LIN {X 0,Y 573.286,Z 595.539,A -85,B 0,C 180,E1 -2259.17,E2 -2259.17} C_VEL
LIN {X 0,Y 573.423,Z 585.099,A -85,B 0,C 180,E1 -2260.058,E2 -2260.058} C_VEL
LIN {X 0,Y 573.528,Z 573.355,A -85,B 0,C 180,E1 -2260.858,E2 -2260.858} C_VEL
LIN {X 0,Y 573.653,Z 562.283,A -85,B 0,C 180,E1 -2261.447,E2 -2261.447} C_VEL
LIN {X 0,Y 573.745,Z 549.174,A -85,B 0,C 180,E1 -2261.974,E2 -2261.974} C_VEL
LIN {X 0,Y 573.879,Z 536.521,A -85,B 0,C 180,E1 -2262.33,E2 -2262.33} C_VEL
LIN {X 0,Y 573.903,Z 523.313,A -85,B 0,C 180,E1 -2262.554,E2 -2262.554} C_VEL
LIN {X 0,Y 573.944,Z 426.723,A -85,B 0,C 180,E1 -2263.769,E2 -2263.769} C_VEL
LIN {X 0,Y 573.378,Z 422.884,A -85,B 0,C 180,E1 -2263.851,E2 -2263.851} C_VEL
LIN {X 0,Y 573.54,Z 403.262,A -85,B 0,C 180,E1 -2266.723,E2 -2266.723} C_VEL
LIN {X 0,Y 573.712,Z 385.787,A -85,B 0,C 180,E1 -2269.314,E2 -2269.314} C_VEL
LIN {X 0,Y 573.994,Z 368.402,A -85,B 0,C 180,E1 -2271.928,E2 -2271.928} C_VEL
LIN {X 0,Y 573.681,Z 364.676,A -85,B 0,C 180,E1 -2272.509,E2 -2272.509} C_VEL
LIN {X 0,Y 573.261,Z 362.581,A -85,B 0,C 180,E1 -2272.86,E2 -2272.86} C_VEL
LIN {X 0,Y 573.259,Z 362.579,A -85,B 0,C 180,E1 -2275.41,E2 -2275.41} C_VEL
LIN {X 0,Y 573.254,Z 362.574,A -85,B 0,C 180,E1 -2278.029,E2 -2278.029} C_VEL
LIN {X 0,Y 573.242,Z 362.58,A -85,B 0,C 180,E1 -2280.884,E2 -2280.884} C_VEL
LIN {X 0,Y 573.265,Z 362.574,A -85,B 0,C 180,E1 -2283.524,E2 -2283.524} C_VEL
LIN {X 0,Y 573.219,Z 362.577,A -85,B 0,C 180,E1 -2286.051,E2 -2286.051} C_VEL
LIN {X 0,Y 573.252,Z 362.577,A -85,B 0,C 180,E1 -2288.701,E2 -2288.701} C_VEL
LIN {X 0,Y 573.232,Z 362.578,A -85,B 0,C 180,E1 -2291.457,E2 -2291.457} C_VEL
LIN {X 0,Y 573.238,Z 362.576,A -85,B 0,C 180,E1 -2294.333,E2 -2294.333} C_VEL
LIN {X 0,Y 573.247,Z 362.576,A -85,B 0,C 180,E1 -2297.358,E2 -2297.358} C_VEL
LIN {X 0,Y 573.242,Z 362.577,A -85,B 0,C 180,E1 -2300.392,E2 -2300.392} C_VEL
LIN {X 0,Y 573.255,Z 362.577,A -85,B 0,C 180,E1 -2303.078,E2 -2303.078} C_VEL
LIN {X 0,Y 573.269,Z 362.57,A -85,B 0,C 180,E1 -2305.671,E2 -2305.671} C_VEL
LIN {X 0,Y 573.244,Z 362.576,A -85,B 0,C 180,E1 -2308.185,E2 -2308.185} C_VEL
LIN {X 0,Y 573.267,Z 362.58,A -85,B 0,C 180,E1 -2310.634,E2 -2310.634} C_VEL
LIN {X 0,Y 573.254,Z 362.576,A -85,B 0,C 180,E1 -2313.024,E2 -2313.024} C_VEL
LIN {X 0,Y 573.278,Z 362.57,A -85,B 0,C 180,E1 -2315.366,E2 -2315.366} C_VEL
LIN {X 0,Y 573.233,Z 362.583,A -85,B 0,C 180,E1 -2318.419,E2 -2318.419} C_VEL
LIN {X 0,Y 573.282,Z 362.575,A -85,B 0,C 180,E1 -2320.728,E2 -2320.728} C_VEL
LIN {X 0,Y 573.253,Z 362.573,A -85,B 0,C 180,E1 -2323.622,E2 -2323.622} C_VEL
LIN {X 0,Y 573.276,Z 362.571,A -85,B 0,C 180,E1 -2325.807,E2 -2325.807} C_VEL
LIN {X 0,Y 573.267,Z 362.575,A -85,B 0,C 180,E1 -2328.745,E2 -2328.745} C_VEL
LIN {X 0,Y 573.259,Z 362.572,A -85,B 0,C 180,E1 -2331.54,E2 -2331.54} C_VEL
LIN {X 0,Y 573.247,Z 362.574,A -85,B 0,C 180,E1 -2333.665,E2 -2333.665} C_VEL
LIN {X 0,Y 573.228,Z 362.578,A -85,B 0,C 180,E1 -2335.781,E2 -2335.781} C_VEL
LIN {X 0,Y 573.31,Z 362.57,A -85,B 0,C 180,E1 -2337.892,E2 -2337.892} C_VEL
LIN {X 0,Y 573.335,Z 362.565,A -85,B 0,C 180,E1 -2340.702,E2 -2340.702} C_VEL
LIN {X 0,Y 573.238,Z 362.575,A -85,B 0,C 180,E1 -2343.515,E2 -2343.515} C_VEL
LIN {X 0,Y 573.293,Z 362.57,A -85,B 0,C 180,E1 -2345.628,E2 -2345.628} C_VEL
LIN {X 0,Y 573.288,Z 362.572,A -85,B 0,C 180,E1 -2348.46,E2 -2348.46} C_VEL
LIN {X 0,Y 573.276,Z 362.57,A -85,B 0,C 180,E1 -2351.312,E2 -2351.312} C_VEL
LIN {X 0,Y 573.286,Z 362.572,A -85,B 0,C 180,E1 -2354.425,E2 -2354.425} C_VEL
LIN {X 0,Y 573.264,Z 362.571,A -85,B 0,C 180,E1 -2357.112,E2 -2357.112} C_VEL
LIN {X 0,Y 573.256,Z 362.579,A -85,B 0,C 180,E1 -2360.077,E2 -2360.077} C_VEL
LIN {X 0,Y 573.238,Z 362.575,A -85,B 0,C 180,E1 -2363.099,E2 -2363.099} C_VEL
LIN {X 0,Y 573.255,Z 362.574,A -85,B 0,C 180,E1 -2364.388,E2 -2364.388} C_VEL
LIN {X 0,Y 572.626,Z 362.652,A -85,B 0,C 180,E1 -2364.974,E2 -2364.974} C_VEL
LIN {X 0,Y 569.779,Z 363.013,A -85,B 0,C 180,E1 -2365.926,E2 -2365.926} C_VEL
LIN {X 0,Y 567.347,Z 363.315,A -85,B 0,C 180,E1 -2366.691,E2 -2366.691} C_VEL
LIN {X 0,Y 566.297,Z 363.442,A -85,B 0,C 180,E1 -2367.282,E2 -2367.282} C_VEL
LIN {X 0,Y 566.211,Z 363.452,A -85,B 0,C 180,E1 -2367.483,E2 -2367.483} C_VEL
LIN {X 0,Y 566.206,Z 363.46,A -85,B 0,C 180,E1 -2369.769,E2 -2369.769} C_VEL
LIN {X 0,Y 566.21,Z 363.45,A -85,B 0,C 180,E1 -2372.43,E2 -2372.43} C_VEL
LIN {X 0,Y 566.205,Z 363.451,A -85,B 0,C 180,E1 -2374.993,E2 -2374.993} C_VEL
LIN {X 0,Y 566.2,Z 363.458,A -85,B 0,C 180,E1 -2377.461,E2 -2377.461} C_VEL
LIN {X 0,Y 566.21,Z 363.451,A -85,B 0,C 180,E1 -2380.199,E2 -2380.199} C_VEL
LIN {X 0,Y 566.209,Z 363.453,A -85,B 0,C 180,E1 -2383.054,E2 -2383.054} C_VEL
LIN {X 0,Y 566.202,Z 363.453,A -85,B 0,C 180,E1 -2386.049,E2 -2386.049} C_VEL
LIN {X 0,Y 566.223,Z 363.454,A -85,B 0,C 180,E1 -2389.213,E2 -2389.213} C_VEL
LIN {X 0,Y 566.193,Z 363.458,A -85,B 0,C 180,E1 -2391.637,E2 -2391.637} C_VEL
LIN {X 0,Y 566.216,Z 363.449,A -85,B 0,C 180,E1 -2394.312,E2 -2394.312} C_VEL
LIN {X 0,Y 566.223,Z 363.451,A -85,B 0,C 180,E1 -2396.898,E2 -2396.898} C_VEL
LIN {X 0,Y 566.185,Z 363.461,A -85,B 0,C 180,E1 -2399.407,E2 -2399.407} C_VEL
LIN {X 0,Y 566.215,Z 363.451,A -85,B 0,C 180,E1 -2401.858,E2 -2401.858} C_VEL
LIN {X 0,Y 566.217,Z 363.45,A -85,B 0,C 180,E1 -2404.251,E2 -2404.251} C_VEL
LIN {X 0,Y 566.173,Z 363.459,A -85,B 0,C 180,E1 -2406.719,E2 -2406.719} C_VEL
LIN {X 0,Y 566.248,Z 363.457,A -85,B 0,C 180,E1 -2409.83,E2 -2409.83} C_VEL
LIN {X 0,Y 566.611,Z 367.185,A -85,B 0,C 180,E1 -2410.506,E2 -2410.506} C_VEL
LIN {X 0,Y 566.454,Z 382.099,A -85,B 0,C 180,E1 -2413.118,E2 -2413.118} C_VEL
LIN {X 0,Y 566.278,Z 399.018,A -85,B 0,C 180,E1 -2416.041,E2 -2416.041} C_VEL
LIN {X 0,Y 567.193,Z 405.355,A -85,B 0,C 180,E1 -2416.155,E2 -2416.155} C_VEL
LIN {X 0,Y 566.949,Z 505.972,A -85,B 0,C 180,E1 -2417.448,E2 -2417.448} C_VEL
LIN {X 0,Y 566.829,Z 519.227,A -85,B 0,C 180,E1 -2417.764,E2 -2417.764} C_VEL
LIN {X 0,Y 566.742,Z 531.382,A -85,B 0,C 180,E1 -2418.194,E2 -2418.194} C_VEL
LIN {X 0,Y 566.604,Z 543.662,A -85,B 0,C 180,E1 -2418.781,E2 -2418.781} C_VEL
LIN {X 0,Y 566.432,Z 555.848,A -85,B 0,C 180,E1 -2419.545,E2 -2419.545} C_VEL
LIN {X 0,Y 566.3,Z 566.133,A -85,B 0,C 180,E1 -2420.355,E2 -2420.355} C_VEL
LIN {X 0,Y 566.183,Z 575.38,A -85,B 0,C 180,E1 -2421.254,E2 -2421.254} C_VEL
LIN {X 0,Y 566.081,Z 584.35,A -85,B 0,C 180,E1 -2422.33,E2 -2422.33} C_VEL
LIN {X 0,Y 566.009,Z 591.459,A -85,B 0,C 180,E1 -2423.386,E2 -2423.386} C_VEL
LIN {X 0,Y 566.004,Z 596.452,A -85,B 0,C 180,E1 -2424.299,E2 -2424.299} C_VEL
LIN {X 0,Y 565.933,Z 601.193,A -85,B 0,C 180,E1 -2425.37,E2 -2425.37} C_VEL
LIN {X 0,Y 565.927,Z 604.826,A -85,B 0,C 180,E1 -2426.44,E2 -2426.44} C_VEL
LIN {X 0,Y 565.877,Z 606.703,A -85,B 0,C 180,E1 -2427.153,E2 -2427.153} C_VEL
LIN {X 0,Y 565.84,Z 608.128,A -85,B 0,C 180,E1 -2427.865,E2 -2427.865} C_VEL
LIN {X 0,Y 565.841,Z 609.756,A -85,B 0,C 180,E1 -2429.288,E2 -2429.288} C_VEL
LIN {X 0,Y 565.839,Z 609.996,A -85,B 0,C 180,E1 -2430,E2 -2430} C_VEL
LIN {X 0,Y 565.841,Z 609.815,A -85,B 0,C 180,E1 -2430.712,E2 -2430.712} C_VEL
LIN {X 0,Y 565.841,Z 608.268,A -85,B 0,C 180,E1 -2432.136,E2 -2432.136} C_VEL
LIN {X 0,Y 565.878,Z 606.907,A -85,B 0,C 180,E1 -2432.848,E2 -2432.848} C_VEL
LIN {X 0,Y 565.927,Z 604.029,A -85,B 0,C 180,E1 -2433.917,E2 -2433.917} C_VEL
LIN {X 0,Y 565.878,Z 600.128,A -85,B 0,C 180,E1 -2434.988,E2 -2434.988} C_VEL
LIN {X 0,Y 565.99,Z 595.096,A -85,B 0,C 180,E1 -2436.059,E2 -2436.059} C_VEL
LIN {X 0,Y 566.031,Z 588.771,A -85,B 0,C 180,E1 -2437.133,E2 -2437.133} C_VEL
LIN {X 0,Y 566.128,Z 580.848,A -85,B 0,C 180,E1 -2438.208,E2 -2438.208} C_VEL
LIN {X 0,Y 566.249,Z 570.997,A -85,B 0,C 180,E1 -2439.285,E2 -2439.285} C_VEL
LIN {X 0,Y 566.42,Z 560.677,A -85,B 0,C 180,E1 -2440.184,E2 -2440.184} C_VEL
LIN {X 0,Y 566.573,Z 549.359,A -85,B 0,C 180,E1 -2440.974,E2 -2440.974} C_VEL
LIN {X 0,Y 566.689,Z 538.183,A -85,B 0,C 180,E1 -2441.592,E2 -2441.592} C_VEL
LIN {X 0,Y 566.78,Z 525.588,A -85,B 0,C 180,E1 -2442.119,E2 -2442.119} C_VEL
LIN {X 0,Y 566.933,Z 512.409,A -85,B 0,C 180,E1 -2442.507,E2 -2442.507} C_VEL
LIN {X 0,Y 566.986,Z 500.032,A -85,B 0,C 180,E1 -2442.733,E2 -2442.733} C_VEL
LIN {X 0,Y 567.094,Z 404.105,A -85,B 0,C 180,E1 -2443.954,E2 -2443.954} C_VEL
LIN {X 0,Y 566.267,Z 399.007,A -85,B 0,C 180,E1 -2444.052,E2 -2444.052} C_VEL
LIN {X 0,Y 566.431,Z 382.626,A -85,B 0,C 180,E1 -2446.881,E2 -2446.881} C_VEL
LIN {X 0,Y 566.614,Z 367.284,A -85,B 0,C 180,E1 -2449.566,E2 -2449.566} C_VEL
LIN {X 0,Y 566.238,Z 363.454,A -85,B 0,C 180,E1 -2450.289,E2 -2450.289} C_VEL
LIN {X 0,Y 566.174,Z 363.461,A -85,B 0,C 180,E1 -2453.281,E2 -2453.281} C_VEL
LIN {X 0,Y 566.217,Z 363.451,A -85,B 0,C 180,E1 -2455.749,E2 -2455.749} C_VEL
LIN {X 0,Y 566.207,Z 363.451,A -85,B 0,C 180,E1 -2458.202,E2 -2458.202} C_VEL
LIN {X 0,Y 566.195,Z 363.457,A -85,B 0,C 180,E1 -2461.076,E2 -2461.076} C_VEL
LIN {X 0,Y 566.217,Z 363.449,A -85,B 0,C 180,E1 -2463.734,E2 -2463.734} C_VEL
LIN {X 0,Y 566.204,Z 363.458,A -85,B 0,C 180,E1 -2466.57,E2 -2466.57} C_VEL
LIN {X 0,Y 566.22,Z 363.448,A -85,B 0,C 180,E1 -2469.686,E2 -2469.686} C_VEL
LIN {X 0,Y 566.206,Z 363.455,A -85,B 0,C 180,E1 -2472.917,E2 -2472.917} C_VEL
LIN {X 0,Y 566.208,Z 363.453,A -85,B 0,C 180,E1 -2476.048,E2 -2476.048} C_VEL
LIN {X 0,Y 566.188,Z 363.457,A -85,B 0,C 180,E1 -2478.861,E2 -2478.861} C_VEL
LIN {X 0,Y 566.188,Z 363.453,A -85,B 0,C 180,E1 -2481.637,E2 -2481.637} C_VEL
LIN {X 0,Y 566.167,Z 363.463,A -85,B 0,C 180,E1 -2484.308,E2 -2484.308} C_VEL
LIN {X 0,Y 566.226,Z 363.45,A -85,B 0,C 180,E1 -2486.898,E2 -2486.898} C_VEL
LIN {X 0,Y 566.186,Z 363.453,A -85,B 0,C 180,E1 -2489.407,E2 -2489.407} C_VEL
LIN {X 0,Y 566.217,Z 363.452,A -85,B 0,C 180,E1 -2491.858,E2 -2491.858} C_VEL
LIN {X 0,Y 566.221,Z 363.459,A -85,B 0,C 180,E1 -2494.251,E2 -2494.251} C_VEL
LIN {X 0,Y 566.175,Z 363.456,A -85,B 0,C 180,E1 -2496.719,E2 -2496.719} C_VEL
LIN {X 0,Y 566.219,Z 363.451,A -85,B 0,C 180,E1 -2499.663,E2 -2499.663} C_VEL
LIN {X 0,Y 566.209,Z 363.452,A -85,B 0,C 180,E1 -2502.669,E2 -2502.669} C_VEL
LIN {X 0,Y 566.241,Z 363.449,A -85,B 0,C 180,E1 -2505.627,E2 -2505.627} C_VEL
LIN {X 0,Y 566.241,Z 363.447,A -85,B 0,C 180,E1 -2508.675,E2 -2508.675} C_VEL
LIN {X 0,Y 566.233,Z 363.449,A -85,B 0,C 180,E1 -2511.434,E2 -2511.434} C_VEL
LIN {X 0,Y 566.264,Z 363.447,A -85,B 0,C 180,E1 -2514.302,E2 -2514.302} C_VEL
LIN {X 0,Y 566.286,Z 363.451,A -85,B 0,C 180,E1 -2517.866,E2 -2517.866} C_VEL
LIN {X 0,Y 566.306,Z 363.438,A -85,B 0,C 180,E1 -2520.711,E2 -2520.711} C_VEL
LIN {X 0,Y 566.278,Z 363.441,A -85,B 0,C 180,E1 -2522.846,E2 -2522.846} C_VEL
LIN {X 0,Y 566.263,Z 363.453,A -85,B 0,C 180,E1 -2525.698,E2 -2525.698} C_VEL
LIN {X 0,Y 566.211,Z 363.45,A -85,B 0,C 180,E1 -2528.566,E2 -2528.566} C_VEL
LIN {X 0,Y 566.248,Z 363.452,A -85,B 0,C 180,E1 -2531.454,E2 -2531.454} C_VEL
LIN {X 0,Y 566.24,Z 363.446,A -85,B 0,C 180,E1 -2534.506,E2 -2534.506} C_VEL
LIN {X 0,Y 566.204,Z 363.457,A -85,B 0,C 180,E1 -2537.332,E2 -2537.332} C_VEL
LIN {X 0,Y 566.218,Z 363.449,A -85,B 0,C 180,E1 -2540.337,E2 -2540.337} C_VEL
LIN {X 0,Y 566.176,Z 363.461,A -85,B 0,C 180,E1 -2543.281,E2 -2543.281} C_VEL
LIN {X 0,Y 566.215,Z 363.454,A -85,B 0,C 180,E1 -2545.749,E2 -2545.749} C_VEL
LIN {X 0,Y 566.208,Z 363.45,A -85,B 0,C 180,E1 -2548.202,E2 -2548.202} C_VEL
LIN {X 0,Y 566.195,Z 363.457,A -85,B 0,C 180,E1 -2551.076,E2 -2551.076} C_VEL
LIN {X 0,Y 566.201,Z 363.454,A -85,B 0,C 180,E1 -2553.732,E2 -2553.732} C_VEL
LIN {X 0,Y 566.204,Z 363.452,A -85,B 0,C 180,E1 -2556.57,E2 -2556.57} C_VEL
LIN {X 0,Y 566.217,Z 363.451,A -85,B 0,C 180,E1 -2559.685,E2 -2559.685} C_VEL
LIN {X 0,Y 566.207,Z 363.456,A -85,B 0,C 180,E1 -2562.917,E2 -2562.917} C_VEL
LIN {X 0,Y 566.198,Z 363.451,A -85,B 0,C 180,E1 -2566.049,E2 -2566.049} C_VEL
LIN {X 0,Y 566.208,Z 363.457,A -85,B 0,C 180,E1 -2569.214,E2 -2569.214} C_VEL
LIN {X 0,Y 566.194,Z 363.453,A -85,B 0,C 180,E1 -2571.637,E2 -2571.637} C_VEL
LIN {X 0,Y 566.178,Z 363.455,A -85,B 0,C 180,E1 -2574.309,E2 -2574.309} C_VEL
LIN {X 0,Y 566.224,Z 363.458,A -85,B 0,C 180,E1 -2576.898,E2 -2576.898} C_VEL
LIN {X 0,Y 566.192,Z 363.455,A -85,B 0,C 180,E1 -2579.408,E2 -2579.408} C_VEL
LIN {X 0,Y 566.216,Z 363.45,A -85,B 0,C 180,E1 -2581.857,E2 -2581.857} C_VEL
LIN {X 0,Y 566.219,Z 363.453,A -85,B 0,C 180,E1 -2584.251,E2 -2584.251} C_VEL
LIN {X 0,Y 566.208,Z 363.538,A -85,B 0,C 180,E1 -2587.024,E2 -2587.024} C_VEL
LIN {X 0,Y 567.015,Z 368.31,A -85,B 0,C 180,E1 -2587.787,E2 -2587.787} C_VEL
LIN {X 0,Y 566.782,Z 385.899,A -85,B 0,C 180,E1 -2590.457,E2 -2590.457} C_VEL
LIN {X 0,Y 566.557,Z 404.552,A -85,B 0,C 180,E1 -2593.258,E2 -2593.258} C_VEL
LIN {X 0,Y 566.39,Z 423.124,A -85,B 0,C 180,E1 -2595.997,E2 -2595.997} C_VEL
LIN {X 0,Y 567.197,Z 428.387,A -85,B 0,C 180,E1 -2596.085,E2 -2596.085} C_VEL
LIN {X 0,Y 566.968,Z 530.935,A -85,B 0,C 180,E1 -2597.403,E2 -2597.403} C_VEL
LIN {X 0,Y 566.852,Z 544.211,A -85,B 0,C 180,E1 -2597.719,E2 -2597.719} C_VEL
LIN {X 0,Y 566.759,Z 556.37,A -85,B 0,C 180,E1 -2598.148,E2 -2598.148} C_VEL
LIN {X 0,Y 566.59,Z 568.445,A -85,B 0,C 180,E1 -2598.724,E2 -2598.724} C_VEL
LIN {X 0,Y 566.442,Z 580.196,A -85,B 0,C 180,E1 -2599.455,E2 -2599.455} C_VEL
LIN {X 0,Y 566.321,Z 590.599,A -85,B 0,C 180,E1 -2600.265,E2 -2600.265} C_VEL
LIN {X 0,Y 566.207,Z 599.111,A -85,B 0,C 180,E1 -2601.074,E2 -2601.074} C_VEL
LIN {X 0,Y 566.112,Z 606.959,A -85,B 0,C 180,E1 -2601.971,E2 -2601.971} C_VEL
LIN {X 0,Y 566.004,Z 614.621,A -85,B 0,C 180,E1 -2603.046,E2 -2603.046} C_VEL
LIN {X 0,Y 566.004,Z 621.679,A -85,B 0,C 180,E1 -2604.299,E2 -2604.299} C_VEL
LIN {X 0,Y 565.933,Z 626.372,A -85,B 0,C 180,E1 -2605.37,E2 -2605.37} C_VEL
LIN {X 0,Y 565.927,Z 629.957,A -85,B 0,C 180,E1 -2606.44,E2 -2606.44} C_VEL
LIN {X 0,Y 565.878,Z 631.808,A -85,B 0,C 180,E1 -2607.152,E2 -2607.152} C_VEL
LIN {X 0,Y 565.846,Z 634.185,A -85,B 0,C 180,E1 -2608.576,E2 -2608.576} C_VEL
LIN {X 0,Y 565.839,Z 635,A -85,B 0,C 180,E1 -2610,E2 -2610} C_VEL
LIN {X 0,Y 565.846,Z 634.186,A -85,B 0,C 180,E1 -2611.423,E2 -2611.423} C_VEL
LIN {X 0,Y 565.878,Z 631.81,A -85,B 0,C 180,E1 -2612.847,E2 -2612.847} C_VEL
LIN {X 0,Y 565.926,Z 628.896,A -85,B 0,C 180,E1 -2613.916,E2 -2613.916} C_VEL
LIN {X 0,Y 565.878,Z 624.949,A -85,B 0,C 180,E1 -2614.987,E2 -2614.987} C_VEL
LIN {X 0,Y 566.002,Z 619.867,A -85,B 0,C 180,E1 -2616.058,E2 -2616.058} C_VEL
LIN {X 0,Y 566.04,Z 613.469,A -85,B 0,C 180,E1 -2617.132,E2 -2617.132} C_VEL
LIN {X 0,Y 566.133,Z 605.479,A -85,B 0,C 180,E1 -2618.208,E2 -2618.208} C_VEL
LIN {X 0,Y 566.228,Z 597.336,A -85,B 0,C 180,E1 -2619.105,E2 -2619.105} C_VEL
LIN {X 0,Y 566.343,Z 587.401,A -85,B 0,C 180,E1 -2620.005,E2 -2620.005} C_VEL
LIN {X 0,Y 566.529,Z 576.292,A -85,B 0,C 180,E1 -2620.807,E2 -2620.807} C_VEL
LIN {X 0,Y 566.612,Z 565.177,A -85,B 0,C 180,E1 -2621.447,E2 -2621.447} C_VEL
LIN {X 0,Y 566.737,Z 552.984,A -85,B 0,C 180,E1 -2621.988,E2 -2621.988} C_VEL
LIN {X 0,Y 566.9,Z 540.178,A -85,B 0,C 180,E1 -2622.394,E2 -2622.394} C_VEL
LIN {X 0,Y 566.977,Z 526.605,A -85,B 0,C 180,E1 -2622.665,E2 -2622.665} C_VEL
LIN {X 0,Y 567.036,Z 427.418,A -85,B 0,C 180,E1 -2623.932,E2 -2623.932} C_VEL
LIN {X 0,Y 566.377,Z 422.884,A -85,B 0,C 180,E1 -2624.026,E2 -2624.026} C_VEL
LIN {X 0,Y 566.568,Z 402.098,A -85,B 0,C 180,E1 -2627.109,E2 -2627.109} C_VEL
LIN {X 0,Y 566.796,Z 384.545,A -85,B 0,C 180,E1 -2629.748,E2 -2629.748} C_VEL
LIN {X 0,Y 567.018,Z 368.321,A -85,B 0,C 180,E1 -2632.212,E2 -2632.212} C_VEL
LIN {X 0,Y 566.209,Z 363.46,A -85,B 0,C 180,E1 -2632.998,E2 -2632.998} C_VEL
LIN {X 0,Y 566.218,Z 363.452,A -85,B 0,C 180,E1 -2635.749,E2 -2635.749} C_VEL
LIN {X 0,Y 566.205,Z 363.452,A -85,B 0,C 180,E1 -2638.202,E2 -2638.202} C_VEL
LIN {X 0,Y 566.203,Z 363.46,A -85,B 0,C 180,E1 -2641.078,E2 -2641.078} C_VEL
LIN {X 0,Y 566.215,Z 363.45,A -85,B 0,C 180,E1 -2643.734,E2 -2643.734} C_VEL
LIN {X 0,Y 566.203,Z 363.453,A -85,B 0,C 180,E1 -2646.57,E2 -2646.57} C_VEL
LIN {X 0,Y 566.225,Z 363.453,A -85,B 0,C 180,E1 -2649.273,E2 -2649.273} C_VEL
LIN {X 0,Y 566.192,Z 363.452,A -85,B 0,C 180,E1 -2652.09,E2 -2652.09} C_VEL
LIN {X 0,Y 566.177,Z 363.462,A -85,B 0,C 180,E1 -2655.036,E2 -2655.036} C_VEL
LIN {X 0,Y 566.214,Z 363.449,A -85,B 0,C 180,E1 -2657.913,E2 -2657.913} C_VEL
LIN {X 0,Y 566.217,Z 363.457,A -85,B 0,C 180,E1 -2660.726,E2 -2660.726} C_VEL
LIN {X 0,Y 566.186,Z 363.453,A -85,B 0,C 180,E1 -2663.788,E2 -2663.788} C_VEL
LIN {X 0,Y 566.214,Z 363.452,A -85,B 0,C 180,E1 -2666.266,E2 -2666.266} C_VEL
LIN {X 0,Y 566.194,Z 363.458,A -85,B 0,C 180,E1 -2668.924,E2 -2668.924} C_VEL
LIN {X 0,Y 566.215,Z 363.45,A -85,B 0,C 180,E1 -2671.857,E2 -2671.857} C_VEL
LIN {X 0,Y 566.216,Z 363.453,A -85,B 0,C 180,E1 -2674.251,E2 -2674.251} C_VEL
LIN {X 0,Y 566.175,Z 363.462,A -85,B 0,C 180,E1 -2676.718,E2 -2676.718} C_VEL
LIN {X 0,Y 566.216,Z 363.449,A -85,B 0,C 180,E1 -2679.663,E2 -2679.663} C_VEL
LIN {X 0,Y 566.202,Z 363.458,A -85,B 0,C 180,E1 -2682.668,E2 -2682.668} C_VEL
LIN {X 0,Y 566.237,Z 363.447,A -85,B 0,C 180,E1 -2685.627,E2 -2685.627} C_VEL
LIN {X 0,Y 566.239,Z 363.451,A -85,B 0,C 180,E1 -2688.675,E2 -2688.675} C_VEL
LIN {X 0,Y 566.209,Z 363.45,A -85,B 0,C 180,E1 -2691.434,E2 -2691.434} C_VEL
LIN {X 0,Y 566.259,Z 363.454,A -85,B 0,C 180,E1 -2694.302,E2 -2694.302} C_VEL
LIN {X 0,Y 566.282,Z 363.445,A -85,B 0,C 180,E1 -2697.866,E2 -2697.866} C_VEL
LIN {X 0,Y 566.305,Z 363.44,A -85,B 0,C 180,E1 -2700.711,E2 -2700.711} C_VEL
LIN {X 0,Y 566.277,Z 363.442,A -85,B 0,C 180,E1 -2702.846,E2 -2702.846} C_VEL
LIN {X 0,Y 566.261,Z 363.447,A -85,B 0,C 180,E1 -2705.698,E2 -2705.698} C_VEL
LIN {X 0,Y 566.231,Z 363.45,A -85,B 0,C 180,E1 -2708.566,E2 -2708.566} C_VEL
LIN {X 0,Y 566.246,Z 363.447,A -85,B 0,C 180,E1 -2711.454,E2 -2711.454} C_VEL
LIN {X 0,Y 566.239,Z 363.448,A -85,B 0,C 180,E1 -2714.507,E2 -2714.507} C_VEL
LIN {X 0,Y 566.208,Z 363.452,A -85,B 0,C 180,E1 -2717.331,E2 -2717.331} C_VEL
LIN {X 0,Y 566.217,Z 363.452,A -85,B 0,C 180,E1 -2720.337,E2 -2720.337} C_VEL
LIN {X 0,Y 566.193,Z 363.455,A -85,B 0,C 180,E1 -2723.404,E2 -2723.404} C_VEL
LIN {X 0,Y 566.22,Z 363.458,A -85,B 0,C 180,E1 -2725.749,E2 -2725.749} C_VEL
LIN {X 0,Y 566.211,Z 363.452,A -85,B 0,C 180,E1 -2727.483,E2 -2727.483} C_VEL
LIN {X 0,Y 565.538,Z 363.539,A -85,B 0,C 180,E1 -2728.076,E2 -2728.076} C_VEL
LIN {X 0,Y 562.671,Z 363.892,A -85,B 0,C 180,E1 -2729.04,E2 -2729.04} C_VEL
LIN {X 0,Y 560.256,Z 364.2,A -85,B 0,C 180,E1 -2729.815,E2 -2729.815} C_VEL
LIN {X 0,Y 559.226,Z 364.322,A -85,B 0,C 180,E1 -2730.414,E2 -2730.414} C_VEL
LIN {X 0,Y 559.146,Z 364.33,A -85,B 0,C 180,E1 -2730.617,E2 -2730.617} C_VEL
LIN {X 0,Y 559.168,Z 364.335,A -85,B 0,C 180,E1 -2733.575,E2 -2733.575} C_VEL
LIN {X 0,Y 559.171,Z 364.327,A -85,B 0,C 180,E1 -2736.448,E2 -2736.448} C_VEL
LIN {X 0,Y 559.178,Z 364.327,A -85,B 0,C 180,E1 -2738.934,E2 -2738.934} C_VEL
LIN {X 0,Y 559.181,Z 364.327,A -85,B 0,C 180,E1 -2742.138,E2 -2742.138} C_VEL
LIN {X 0,Y 559.144,Z 364.33,A -85,B 0,C 180,E1 -2744.739,E2 -2744.739} C_VEL
LIN {X 0,Y 559.161,Z 364.334,A -85,B 0,C 180,E1 -2747.256,E2 -2747.256} C_VEL
LIN {X 0,Y 559.185,Z 364.326,A -85,B 0,C 180,E1 -2750.135,E2 -2750.135} C_VEL
LIN {X 0,Y 559.15,Z 364.332,A -85,B 0,C 180,E1 -2752.892,E2 -2752.892} C_VEL
LIN {X 0,Y 559.161,Z 364.334,A -85,B 0,C 180,E1 -2755.556,E2 -2755.556} C_VEL
LIN {X 0,Y 559.169,Z 364.327,A -85,B 0,C 180,E1 -2758.137,E2 -2758.137} C_VEL
LIN {X 0,Y 559.146,Z 364.331,A -85,B 0,C 180,E1 -2760.646,E2 -2760.646} C_VEL
LIN {X 0,Y 559.174,Z 364.335,A -85,B 0,C 180,E1 -2763.173,E2 -2763.173} C_VEL
LIN {X 0,Y 559.159,Z 364.335,A -85,B 0,C 180,E1 -2765.495,E2 -2765.495} C_VEL
LIN {X 0,Y 559.175,Z 364.331,A -85,B 0,C 180,E1 -2768.624,E2 -2768.624} C_VEL
LIN {X 0,Y 559.211,Z 364.505,A -85,B 0,C 180,E1 -2769.733,E2 -2769.733} C_VEL
LIN {X 0,Y 559.644,Z 367.893,A -85,B 0,C 180,E1 -2770.365,E2 -2770.365} C_VEL
LIN {X 0,Y 559.447,Z 382.395,A -85,B 0,C 180,E1 -2772.952,E2 -2772.952} C_VEL
LIN {X 0,Y 559.25,Z 399.021,A -85,B 0,C 180,E1 -2775.861,E2 -2775.861} C_VEL
LIN {X 0,Y 560.276,Z 405.401,A -85,B 0,C 180,E1 -2775.981,E2 -2775.981} C_VEL
LIN {X 0,Y 560.047,Z 506,A -85,B 0,C 180,E1 -2777.291,E2 -2777.291} C_VEL
LIN {X 0,Y 559.91,Z 519.245,A -85,B 0,C 180,E1 -2777.61,E2 -2777.61} C_VEL
LIN {X 0,Y 559.786,Z 531.397,A -85,B 0,C 180,E1 -2778.045,E2 -2778.045} C_VEL
LIN {X 0,Y 559.649,Z 543.084,A -85,B 0,C 180,E1 -2778.607,E2 -2778.607} C_VEL
LIN {X 0,Y 559.481,Z 554.564,A -85,B 0,C 180,E1 -2779.322,E2 -2779.322} C_VEL
LIN {X 0,Y 559.307,Z 565.081,A -85,B 0,C 180,E1 -2780.142,E2 -2780.142} C_VEL
LIN {X 0,Y 559.197,Z 573.676,A -85,B 0,C 180,E1 -2780.961,E2 -2780.961} C_VEL
LIN {X 0,Y 559.05,Z 581.596,A -85,B 0,C 180,E1 -2781.87,E2 -2781.87} C_VEL
LIN {X 0,Y 558.971,Z 589.457,A -85,B 0,C 180,E1 -2782.977,E2 -2782.977} C_VEL
LIN {X 0,Y 558.936,Z 596.455,A -85,B 0,C 180,E1 -2784.227,E2 -2784.227} C_VEL
LIN {X 0,Y 558.827,Z 601.195,A -85,B 0,C 180,E1 -2785.311,E2 -2785.311} C_VEL
LIN {X 0,Y 558.836,Z 604.828,A -85,B 0,C 180,E1 -2786.395,E2 -2786.395} C_VEL
LIN {X 0,Y 558.799,Z 606.704,A -85,B 0,C 180,E1 -2787.116,E2 -2787.116} C_VEL
LIN {X 0,Y 558.746,Z 608.128,A -85,B 0,C 180,E1 -2787.838,E2 -2787.838} C_VEL
LIN {X 0,Y 558.741,Z 609.757,A -85,B 0,C 180,E1 -2789.279,E2 -2789.279} C_VEL
LIN {X 0,Y 558.74,Z 609.996,A -85,B 0,C 180,E1 -2790,E2 -2790} C_VEL
LIN {X 0,Y 558.741,Z 609.815,A -85,B 0,C 180,E1 -2790.721,E2 -2790.721} C_VEL
LIN {X 0,Y 558.746,Z 608.266,A -85,B 0,C 180,E1 -2792.163,E2 -2792.163} C_VEL
LIN {X 0,Y 558.8,Z 606.905,A -85,B 0,C 180,E1 -2792.884,E2 -2792.884} C_VEL
LIN {X 0,Y 558.844,Z 604.027,A -85,B 0,C 180,E1 -2793.966,E2 -2793.966} C_VEL
LIN {X 0,Y 558.798,Z 600.126,A -85,B 0,C 180,E1 -2795.051,E2 -2795.051} C_VEL
LIN {X 0,Y 558.91,Z 595.093,A -85,B 0,C 180,E1 -2796.136,E2 -2796.136} C_VEL
LIN {X 0,Y 558.973,Z 588.767,A -85,B 0,C 180,E1 -2797.223,E2 -2797.223} C_VEL
LIN {X 0,Y 559.091,Z 580.843,A -85,B 0,C 180,E1 -2798.312,E2 -2798.312} C_VEL
LIN {X 0,Y 559.224,Z 570.99,A -85,B 0,C 180,E1 -2799.403,E2 -2799.403} C_VEL
LIN {X 0,Y 559.412,Z 560.67,A -85,B 0,C 180,E1 -2800.313,E2 -2800.313} C_VEL
LIN {X 0,Y 559.588,Z 549.687,A -85,B 0,C 180,E1 -2801.091,E2 -2801.091} C_VEL
LIN {X 0,Y 559.725,Z 538.171,A -85,B 0,C 180,E1 -2801.738,E2 -2801.738} C_VEL
LIN {X 0,Y 559.83,Z 525.571,A -85,B 0,C 180,E1 -2802.272,E2 -2802.272} C_VEL
LIN {X 0,Y 560.015,Z 512.385,A -85,B 0,C 180,E1 -2802.664,E2 -2802.664} C_VEL
LIN {X 0,Y 560.088,Z 499.989,A -85,B 0,C 180,E1 -2802.893,E2 -2802.893} C_VEL
LIN {X 0,Y 560.254,Z 405.177,A -85,B 0,C 180,E1 -2804.113,E2 -2804.113} C_VEL
LIN {X 0,Y 559.248,Z 399.003,A -85,B 0,C 180,E1 -2804.232,E2 -2804.232} C_VEL
LIN {X 0,Y 559.438,Z 381.481,A -85,B 0,C 180,E1 -2807.3,E2 -2807.3} C_VEL
LIN {X 0,Y 559.627,Z 367.376,A -85,B 0,C 180,E1 -2809.821,E2 -2809.821} C_VEL
LIN {X 0,Y 559.188,Z 364.333,A -85,B 0,C 180,E1 -2810.412,E2 -2810.412} C_VEL
LIN {X 0,Y 559.143,Z 364.335,A -85,B 0,C 180,E1 -2813.428,E2 -2813.428} C_VEL
LIN {X 0,Y 559.184,Z 364.328,A -85,B 0,C 180,E1 -2816.097,E2 -2816.097} C_VEL
LIN {X 0,Y 559.168,Z 364.332,A -85,B 0,C 180,E1 -2818.53,E2 -2818.53} C_VEL
LIN {X 0,Y 559.15,Z 364.332,A -85,B 0,C 180,E1 -2821.273,E2 -2821.273} C_VEL
LIN {X 0,Y 559.172,Z 364.327,A -85,B 0,C 180,E1 -2823.95,E2 -2823.95} C_VEL
LIN {X 0,Y 559.145,Z 364.333,A -85,B 0,C 180,E1 -2827.109,E2 -2827.109} C_VEL
LIN {X 0,Y 559.166,Z 364.328,A -85,B 0,C 180,E1 -2829.942,E2 -2829.942} C_VEL
LIN {X 0,Y 559.162,Z 364.335,A -85,B 0,C 180,E1 -2832.744,E2 -2832.744} C_VEL
LIN {X 0,Y 559.161,Z 364.328,A -85,B 0,C 180,E1 -2835.761,E2 -2835.761} C_VEL
LIN {X 0,Y 559.194,Z 364.329,A -85,B 0,C 180,E1 -2838.232,E2 -2838.232} C_VEL
LIN {X 0,Y 559.178,Z 364.326,A -85,B 0,C 180,E1 -2841.192,E2 -2841.192} C_VEL
LIN {X 0,Y 559.144,Z 364.331,A -85,B 0,C 180,E1 -2843.789,E2 -2843.789} C_VEL
LIN {X 0,Y 559.168,Z 364.336,A -85,B 0,C 180,E1 -2846.425,E2 -2846.425} C_VEL
LIN {X 0,Y 559.161,Z 364.329,A -85,B 0,C 180,E1 -2848.981,E2 -2848.981} C_VEL
LIN {X 0,Y 559.174,Z 364.327,A -85,B 0,C 180,E1 -2851.619,E2 -2851.619} C_VEL
LIN {X 0,Y 559.188,Z 364.329,A -85,B 0,C 180,E1 -2853.903,E2 -2853.903} C_VEL
LIN {X 0,Y 559.145,Z 364.334,A -85,B 0,C 180,E1 -2856.572,E2 -2856.572} C_VEL
LIN {X 0,Y 559.186,Z 364.325,A -85,B 0,C 180,E1 -2859.396,E2 -2859.396} C_VEL
LIN {X 0,Y 559.155,Z 364.332,A -85,B 0,C 180,E1 -2861.686,E2 -2861.686} C_VEL
LIN {X 0,Y 559.17,Z 364.334,A -85,B 0,C 180,E1 -2863.948,E2 -2863.948} C_VEL
LIN {X 0,Y 559.178,Z 364.333,A -85,B 0,C 180,E1 -2866.184,E2 -2866.184} C_VEL
LIN {X 0,Y 559.201,Z 364.323,A -85,B 0,C 180,E1 -2869.134,E2 -2869.134} C_VEL
LIN {X 0,Y 559.21,Z 364.33,A -85,B 0,C 180,E1 -2872.054,E2 -2872.054} C_VEL
LIN {X 0,Y 559.258,Z 364.316,A -85,B 0,C 180,E1 -2874.953,E2 -2874.953} C_VEL
LIN {X 0,Y 559.257,Z 364.326,A -85,B 0,C 180,E1 -2877.839,E2 -2877.839} C_VEL
LIN {X 0,Y 559.277,Z 364.314,A -85,B 0,C 180,E1 -2880.72,E2 -2880.72} C_VEL
LIN {X 0,Y 559.244,Z 364.318,A -85,B 0,C 180,E1 -2882.881,E2 -2882.881} C_VEL
LIN {X 0,Y 559.233,Z 364.328,A -85,B 0,C 180,E1 -2885.77,E2 -2885.77} C_VEL
LIN {X 0,Y 559.175,Z 364.326,A -85,B 0,C 180,E1 -2888.675,E2 -2888.675} C_VEL
LIN {X 0,Y 559.211,Z 364.331,A -85,B 0,C 180,E1 -2891.6,E2 -2891.6} C_VEL
LIN {X 0,Y 559.206,Z 364.322,A -85,B 0,C 180,E1 -2894.595,E2 -2894.595} C_VEL
LIN {X 0,Y 559.163,Z 364.338,A -85,B 0,C 180,E1 -2897.557,E2 -2897.557} C_VEL
LIN {X 0,Y 559.175,Z 364.331,A -85,B 0,C 180,E1 -2899.837,E2 -2899.837} C_VEL
LIN {X 0,Y 559.147,Z 364.331,A -85,B 0,C 180,E1 -2902.153,E2 -2902.153} C_VEL
LIN {X 0,Y 559.181,Z 364.333,A -85,B 0,C 180,E1 -2905.298,E2 -2905.298} C_VEL
LIN {X 0,Y 559.173,Z 364.326,A -85,B 0,C 180,E1 -2908.381,E2 -2908.381} C_VEL
LIN {X 0,Y 559.151,Z 364.338,A -85,B 0,C 180,E1 -2911.273,E2 -2911.273} C_VEL
LIN {X 0,Y 559.159,Z 364.329,A -85,B 0,C 180,E1 -2913.947,E2 -2913.947} C_VEL
LIN {X 0,Y 559.145,Z 364.338,A -85,B 0,C 180,E1 -2917.108,E2 -2917.108} C_VEL
LIN {X 0,Y 559.164,Z 364.328,A -85,B 0,C 180,E1 -2919.941,E2 -2919.941} C_VEL
LIN {X 0,Y 559.163,Z 364.331,A -85,B 0,C 180,E1 -2922.743,E2 -2922.743} C_VEL
LIN {X 0,Y 559.153,Z 364.33,A -85,B 0,C 180,E1 -2925.761,E2 -2925.761} C_VEL
LIN {X 0,Y 559.166,Z 364.327,A -85,B 0,C 180,E1 -2928.23,E2 -2928.23} C_VEL
LIN {X 0,Y 559.182,Z 364.332,A -85,B 0,C 180,E1 -2931.191,E2 -2931.191} C_VEL
LIN {X 0,Y 559.145,Z 364.33,A -85,B 0,C 180,E1 -2933.789,E2 -2933.789} C_VEL
LIN {X 0,Y 559.167,Z 364.33,A -85,B 0,C 180,E1 -2936.425,E2 -2936.425} C_VEL
LIN {X 0,Y 559.167,Z 364.336,A -85,B 0,C 180,E1 -2938.981,E2 -2938.981} C_VEL
LIN {X 0,Y 559.172,Z 364.328,A -85,B 0,C 180,E1 -2941.619,E2 -2941.619} C_VEL
LIN {X 0,Y 559.186,Z 364.327,A -85,B 0,C 180,E1 -2943.903,E2 -2943.903} C_VEL
LIN {X 0,Y 559.199,Z 364.482,A -85,B 0,C 180,E1 -2946.888,E2 -2946.888} C_VEL
LIN {X 0,Y 560.066,Z 369.428,A -85,B 0,C 180,E1 -2947.691,E2 -2947.691} C_VEL
LIN {X 0,Y 559.811,Z 387.353,A -85,B 0,C 180,E1 -2950.434,E2 -2950.434} C_VEL
LIN {X 0,Y 559.586,Z 403.777,A -85,B 0,C 180,E1 -2952.926,E2 -2952.926} C_VEL
LIN {X 0,Y 559.369,Z 423.124,A -85,B 0,C 180,E1 -2955.818,E2 -2955.818} C_VEL
LIN {X 0,Y 560.303,Z 430.279,A -85,B 0,C 180,E1 -2955.935,E2 -2955.935} C_VEL
LIN {X 0,Y 560.049,Z 530.935,A -85,B 0,C 180,E1 -2957.245,E2 -2957.245} C_VEL
LIN {X 0,Y 559.939,Z 544.21,A -85,B 0,C 180,E1 -2957.565,E2 -2957.565} C_VEL
LIN {X 0,Y 559.809,Z 556.372,A -85,B 0,C 180,E1 -2957.999,E2 -2957.999} C_VEL
LIN {X 0,Y 559.616,Z 568.315,A -85,B 0,C 180,E1 -2958.574,E2 -2958.574} C_VEL
LIN {X 0,Y 559.462,Z 580.194,A -85,B 0,C 180,E1 -2959.322,E2 -2959.322} C_VEL
LIN {X 0,Y 559.302,Z 590.601,A -85,B 0,C 180,E1 -2960.142,E2 -2960.142} C_VEL
LIN {X 0,Y 559.162,Z 599.111,A -85,B 0,C 180,E1 -2960.961,E2 -2960.961} C_VEL
LIN {X 0,Y 559.05,Z 606.959,A -85,B 0,C 180,E1 -2961.869,E2 -2961.869} C_VEL
LIN {X 0,Y 558.944,Z 614.621,A -85,B 0,C 180,E1 -2962.958,E2 -2962.958} C_VEL
LIN {X 0,Y 558.935,Z 621.679,A -85,B 0,C 180,E1 -2964.227,E2 -2964.227} C_VEL
LIN {X 0,Y 558.827,Z 626.372,A -85,B 0,C 180,E1 -2965.311,E2 -2965.311} C_VEL
LIN {X 0,Y 558.836,Z 629.957,A -85,B 0,C 180,E1 -2966.395,E2 -2966.395} C_VEL
LIN {X 0,Y 558.799,Z 631.807,A -85,B 0,C 180,E1 -2967.116,E2 -2967.116} C_VEL
LIN {X 0,Y 558.745,Z 634.184,A -85,B 0,C 180,E1 -2968.558,E2 -2968.558} C_VEL
LIN {X 0,Y 558.74,Z 635,A -85,B 0,C 180,E1 -2970,E2 -2970} C_VEL
LIN {X 0,Y 558.745,Z 634.185,A -85,B 0,C 180,E1 -2971.441,E2 -2971.441} C_VEL
LIN {X 0,Y 558.799,Z 631.81,A -85,B 0,C 180,E1 -2972.884,E2 -2972.884} C_VEL
LIN {X 0,Y 558.843,Z 628.896,A -85,B 0,C 180,E1 -2973.966,E2 -2973.966} C_VEL
LIN {X 0,Y 558.799,Z 624.949,A -85,B 0,C 180,E1 -2975.051,E2 -2975.051} C_VEL
LIN {X 0,Y 558.921,Z 619.867,A -85,B 0,C 180,E1 -2976.135,E2 -2976.135} C_VEL
LIN {X 0,Y 558.977,Z 613.468,A -85,B 0,C 180,E1 -2977.223,E2 -2977.223} C_VEL
LIN {X 0,Y 559.099,Z 605.478,A -85,B 0,C 180,E1 -2978.312,E2 -2978.312} C_VEL
LIN {X 0,Y 559.184,Z 597.335,A -85,B 0,C 180,E1 -2979.221,E2 -2979.221} C_VEL
LIN {X 0,Y 559.356,Z 587.4,A -85,B 0,C 180,E1 -2980.131,E2 -2980.131} C_VEL
LIN {X 0,Y 559.543,Z 576.4,A -85,B 0,C 180,E1 -2980.937,E2 -2980.937} C_VEL
LIN {X 0,Y 559.671,Z 564.461,A -85,B 0,C 180,E1 -2981.628,E2 -2981.628} C_VEL
LIN {X 0,Y 559.82,Z 551.769,A -85,B 0,C 180,E1 -2982.185,E2 -2982.185} C_VEL
LIN {X 0,Y 560.009,Z 538.348,A -85,B 0,C 180,E1 -2982.595,E2 -2982.595} C_VEL
LIN {X 0,Y 560.087,Z 525.088,A -85,B 0,C 180,E1 -2982.846,E2 -2982.846} C_VEL
LIN {X 0,Y 560.189,Z 428.412,A -85,B 0,C 180,E1 -2984.092,E2 -2984.092} C_VEL
LIN {X 0,Y 559.37,Z 422.884,A -85,B 0,C 180,E1 -2984.205,E2 -2984.205} C_VEL
LIN {X 0,Y 559.625,Z 401.877,A -85,B 0,C 180,E1 -2987.361,E2 -2987.361} C_VEL
LIN {X 0,Y 559.947,Z 380.727,A -85,B 0,C 180,E1 -2990.575,E2 -2990.575} C_VEL
LIN {X 0,Y 560.067,Z 369.45,A -85,B 0,C 180,E1 -2992.308,E2 -2992.308} C_VEL
LIN {X 0,Y 559.169,Z 364.337,A -85,B 0,C 180,E1 -2993.149,E2 -2993.149} C_VEL
LIN {X 0,Y 559.185,Z 364.326,A -85,B 0,C 180,E1 -2996.097,E2 -2996.097} C_VEL
LIN {X 0,Y 559.166,Z 364.33,A -85,B 0,C 180,E1 -2998.53,E2 -2998.53} C_VEL
LIN {X 0,Y 559.157,Z 364.336,A -85,B 0,C 180,E1 -3001.275,E2 -3001.275} C_VEL
LIN {X 0,Y 559.17,Z 364.327,A -85,B 0,C 180,E1 -3003.949,E2 -3003.949} C_VEL
LIN {X 0,Y 559.144,Z 364.339,A -85,B 0,C 180,E1 -3007.108,E2 -3007.108} C_VEL
LIN {X 0,Y 559.168,Z 364.327,A -85,B 0,C 180,E1 -3009.942,E2 -3009.942} C_VEL
LIN {X 0,Y 559.16,Z 364.334,A -85,B 0,C 180,E1 -3012.744,E2 -3012.744} C_VEL
LIN {X 0,Y 559.159,Z 364.328,A -85,B 0,C 180,E1 -3015.76,E2 -3015.76} C_VEL
LIN {X 0,Y 559.19,Z 364.326,A -85,B 0,C 180,E1 -3018.232,E2 -3018.232} C_VEL
LIN {X 0,Y 559.177,Z 364.33,A -85,B 0,C 180,E1 -3021.192,E2 -3021.192} C_VEL
LIN {X 0,Y 559.141,Z 364.33,A -85,B 0,C 180,E1 -3023.789,E2 -3023.789} C_VEL
LIN {X 0,Y 559.166,Z 364.332,A -85,B 0,C 180,E1 -3026.425,E2 -3026.425} C_VEL
LIN {X 0,Y 559.158,Z 364.333,A -85,B 0,C 180,E1 -3028.981,E2 -3028.981} C_VEL
LIN {X 0,Y 559.171,Z 364.327,A -85,B 0,C 180,E1 -3031.619,E2 -3031.619} C_VEL
LIN {X 0,Y 559.183,Z 364.326,A -85,B 0,C 180,E1 -3033.903,E2 -3033.903} C_VEL
LIN {X 0,Y 559.145,Z 364.34,A -85,B 0,C 180,E1 -3036.571,E2 -3036.571} C_VEL
LIN {X 0,Y 559.183,Z 364.325,A -85,B 0,C 180,E1 -3039.396,E2 -3039.396} C_VEL
LIN {X 0,Y 559.144,Z 364.33,A -85,B 0,C 180,E1 -3041.686,E2 -3041.686} C_VEL
LIN {X 0,Y 559.169,Z 364.329,A -85,B 0,C 180,E1 -3043.948,E2 -3043.948} C_VEL
LIN {X 0,Y 559.174,Z 364.332,A -85,B 0,C 180,E1 -3046.184,E2 -3046.184} C_VEL
LIN {X 0,Y 559.197,Z 364.324,A -85,B 0,C 180,E1 -3049.134,E2 -3049.134} C_VEL
LIN {X 0,Y 559.199,Z 364.328,A -85,B 0,C 180,E1 -3052.054,E2 -3052.054} C_VEL
LIN {X 0,Y 559.256,Z 364.317,A -85,B 0,C 180,E1 -3054.953,E2 -3054.953} C_VEL
LIN {X 0,Y 559.253,Z 364.32,A -85,B 0,C 180,E1 -3057.839,E2 -3057.839} C_VEL
LIN {X 0,Y 559.276,Z 364.316,A -85,B 0,C 180,E1 -3060.72,E2 -3060.72} C_VEL
LIN {X 0,Y 559.243,Z 364.318,A -85,B 0,C 180,E1 -3062.881,E2 -3062.881} C_VEL
LIN {X 0,Y 559.231,Z 364.323,A -85,B 0,C 180,E1 -3065.77,E2 -3065.77} C_VEL
LIN {X 0,Y 559.19,Z 364.326,A -85,B 0,C 180,E1 -3068.674,E2 -3068.674} C_VEL
LIN {X 0,Y 559.21,Z 364.325,A -85,B 0,C 180,E1 -3071.6,E2 -3071.6} C_VEL
LIN {X 0,Y 559.204,Z 364.324,A -85,B 0,C 180,E1 -3074.596,E2 -3074.596} C_VEL
LIN {X 0,Y 559.167,Z 364.331,A -85,B 0,C 180,E1 -3077.557,E2 -3077.557} C_VEL
LIN {X 0,Y 559.176,Z 364.335,A -85,B 0,C 180,E1 -3079.837,E2 -3079.837} C_VEL
LIN {X 0,Y 559.146,Z 364.335,A -85,B 0,C 180,E1 -3082.153,E2 -3082.153} C_VEL
LIN {X 0,Y 559.183,Z 364.326,A -85,B 0,C 180,E1 -3085.187,E2 -3085.187} C_VEL
LIN {X 0,Y 559.193,Z 364.333,A -85,B 0,C 180,E1 -3087.712,E2 -3087.712} C_VEL
LIN {X 0,Y 559.146,Z 364.33,A -85,B 0,C 180,E1 -3090.617,E2 -3090.617} C_VEL
LIN {X 0,Y 558.486,Z 364.416,A -85,B 0,C 180,E1 -3091.218,E2 -3091.218} C_VEL
LIN {X 0,Y 555.626,Z 364.771,A -85,B 0,C 180,E1 -3092.195,E2 -3092.195} C_VEL
LIN {X 0,Y 553.213,Z 365.07,A -85,B 0,C 180,E1 -3092.98,E2 -3092.98} C_VEL
LIN {X 0,Y 552.192,Z 365.204,A -85,B 0,C 180,E1 -3093.587,E2 -3093.587} C_VEL
LIN {X 0,Y 552.117,Z 365.207,A -85,B 0,C 180,E1 -3093.792,E2 -3093.792} C_VEL
LIN {X 0,Y 552.115,Z 365.206,A -85,B 0,C 180,E1 -3096.747,E2 -3096.747} C_VEL
LIN {X 0,Y 552.133,Z 365.212,A -85,B 0,C 180,E1 -3099.527,E2 -3099.527} C_VEL
LIN {X 0,Y 552.134,Z 365.203,A -85,B 0,C 180,E1 -3102.425,E2 -3102.425} C_VEL
LIN {X 0,Y 552.102,Z 365.216,A -85,B 0,C 180,E1 -3105.563,E2 -3105.563} C_VEL
LIN {X 0,Y 552.135,Z 365.204,A -85,B 0,C 180,E1 -3108.677,E2 -3108.677} C_VEL
LIN {X 0,Y 552.123,Z 365.215,A -85,B 0,C 180,E1 -3111.411,E2 -3111.411} C_VEL
LIN {X 0,Y 552.117,Z 365.206,A -85,B 0,C 180,E1 -3114.159,E2 -3114.159} C_VEL
LIN {X 0,Y 552.119,Z 365.207,A -85,B 0,C 180,E1 -3116.814,E2 -3116.814} C_VEL
LIN {X 0,Y 552.106,Z 365.215,A -85,B 0,C 180,E1 -3119.391,E2 -3119.391} C_VEL
LIN {X 0,Y 552.112,Z 365.207,A -85,B 0,C 180,E1 -3121.902,E2 -3121.902} C_VEL
LIN {X 0,Y 552.159,Z 365.203,A -85,B 0,C 180,E1 -3124.65,E2 -3124.65} C_VEL
LIN {X 0,Y 552.095,Z 365.215,A -85,B 0,C 180,E1 -3127.549,E2 -3127.549} C_VEL
LIN {X 0,Y 552.16,Z 365.289,A -85,B 0,C 180,E1 -3129.584,E2 -3129.584} C_VEL
LIN {X 0,Y 552.65,Z 369.95,A -85,B 0,C 180,E1 -3130.46,E2 -3130.46} C_VEL
LIN {X 0,Y 552.451,Z 384.971,A -85,B 0,C 180,E1 -3133.177,E2 -3133.177} C_VEL
LIN {X 0,Y 552.237,Z 399.236,A -85,B 0,C 180,E1 -3135.69,E2 -3135.69} C_VEL
LIN {X 0,Y 553.414,Z 406.711,A -85,B 0,C 180,E1 -3135.82,E2 -3135.82} C_VEL
LIN {X 0,Y 553.144,Z 506.029,A -85,B 0,C 180,E1 -3137.13,E2 -3137.13} C_VEL
LIN {X 0,Y 552.994,Z 519.263,A -85,B 0,C 180,E1 -3137.453,E2 -3137.453} C_VEL
LIN {X 0,Y 552.837,Z 531.411,A -85,B 0,C 180,E1 -3137.892,E2 -3137.892} C_VEL
LIN {X 0,Y 552.688,Z 542.906,A -85,B 0,C 180,E1 -3138.451,E2 -3138.451} C_VEL
LIN {X 0,Y 552.506,Z 554.57,A -85,B 0,C 180,E1 -3139.186,E2 -3139.186} C_VEL
LIN {X 0,Y 552.305,Z 565.086,A -85,B 0,C 180,E1 -3140.016,E2 -3140.016} C_VEL
LIN {X 0,Y 552.153,Z 573.681,A -85,B 0,C 180,E1 -3140.845,E2 -3140.845} C_VEL
LIN {X 0,Y 552.007,Z 581.6,A -85,B 0,C 180,E1 -3141.765,E2 -3141.765} C_VEL
LIN {X 0,Y 551.895,Z 589.461,A -85,B 0,C 180,E1 -3142.886,E2 -3142.886} C_VEL
LIN {X 0,Y 551.868,Z 596.457,A -85,B 0,C 180,E1 -3144.153,E2 -3144.153} C_VEL
LIN {X 0,Y 551.725,Z 601.198,A -85,B 0,C 180,E1 -3145.251,E2 -3145.251} C_VEL
LIN {X 0,Y 551.75,Z 604.83,A -85,B 0,C 180,E1 -3146.349,E2 -3146.349} C_VEL
LIN {X 0,Y 551.723,Z 606.706,A -85,B 0,C 180,E1 -3147.079,E2 -3147.079} C_VEL
LIN {X 0,Y 551.657,Z 608.128,A -85,B 0,C 180,E1 -3147.81,E2 -3147.81} C_VEL
LIN {X 0,Y 551.642,Z 609.757,A -85,B 0,C 180,E1 -3149.27,E2 -3149.27} C_VEL
LIN {X 0,Y 551.641,Z 609.996,A -85,B 0,C 180,E1 -3150,E2 -3150} C_VEL
LIN {X 0,Y 551.641,Z 609.814,A -85,B 0,C 180,E1 -3150.73,E2 -3150.73} C_VEL
LIN {X 0,Y 551.657,Z 608.264,A -85,B 0,C 180,E1 -3152.19,E2 -3152.19} C_VEL
LIN {X 0,Y 551.724,Z 606.903,A -85,B 0,C 180,E1 -3152.921,E2 -3152.921} C_VEL
LIN {X 0,Y 551.764,Z 604.025,A -85,B 0,C 180,E1 -3154.017,E2 -3154.017} C_VEL
LIN {X 0,Y 551.724,Z 600.124,A -85,B 0,C 180,E1 -3155.116,E2 -3155.116} C_VEL
LIN {X 0,Y 551.811,Z 594.393,A -85,B 0,C 180,E1 -3156.349,E2 -3156.349} C_VEL
LIN {X 0,Y 551.925,Z 587.536,A -85,B 0,C 180,E1 -3157.5,E2 -3157.5} C_VEL
LIN {X 0,Y 552.063,Z 579.353,A -85,B 0,C 180,E1 -3158.603,E2 -3158.603} C_VEL
LIN {X 0,Y 552.197,Z 570.984,A -85,B 0,C 180,E1 -3159.524,E2 -3159.524} C_VEL
LIN {X 0,Y 552.406,Z 560.661,A -85,B 0,C 180,E1 -3160.445,E2 -3160.445} C_VEL
LIN {X 0,Y 552.599,Z 548.861,A -85,B 0,C 180,E1 -3161.286,E2 -3161.286} C_VEL
LIN {X 0,Y 552.769,Z 537.441,A -85,B 0,C 180,E1 -3161.924,E2 -3161.924} C_VEL
LIN {X 0,Y 552.905,Z 525.424,A -85,B 0,C 180,E1 -3162.433,E2 -3162.433} C_VEL
LIN {X 0,Y 553.088,Z 512.362,A -85,B 0,C 180,E1 -3162.825,E2 -3162.825} C_VEL
LIN {X 0,Y 553.194,Z 499.947,A -85,B 0,C 180,E1 -3163.056,E2 -3163.056} C_VEL
LIN {X 0,Y 553.408,Z 406.136,A -85,B 0,C 180,E1 -3164.278,E2 -3164.278} C_VEL
LIN {X 0,Y 552.217,Z 398.949,A -85,B 0,C 180,E1 -3164.426,E2 -3164.426} C_VEL
LIN {X 0,Y 552.437,Z 382.818,A -85,B 0,C 180,E1 -3167.301,E2 -3167.301} C_VEL
LIN {X 0,Y 552.666,Z 369.167,A -85,B 0,C 180,E1 -3169.775,E2 -3169.775} C_VEL
LIN {X 0,Y 552.16,Z 365.209,A -85,B 0,C 180,E1 -3170.538,E2 -3170.538} C_VEL
LIN {X 0,Y 552.103,Z 365.211,A -85,B 0,C 180,E1 -3173.576,E2 -3173.576} C_VEL
LIN {X 0,Y 552.134,Z 365.207,A -85,B 0,C 180,E1 -3175.644,E2 -3175.644} C_VEL
LIN {X 0,Y 552.129,Z 365.209,A -85,B 0,C 180,E1 -3178.562,E2 -3178.562} C_VEL
LIN {X 0,Y 552.115,Z 365.206,A -85,B 0,C 180,E1 -3181.476,E2 -3181.476} C_VEL
LIN {X 0,Y 552.14,Z 365.204,A -85,B 0,C 180,E1 -3184.171,E2 -3184.171} C_VEL
LIN {X 0,Y 552.11,Z 365.215,A -85,B 0,C 180,E1 -3186.747,E2 -3186.747} C_VEL
LIN {X 0,Y 552.135,Z 365.203,A -85,B 0,C 180,E1 -3189.527,E2 -3189.527} C_VEL
LIN {X 0,Y 552.134,Z 365.21,A -85,B 0,C 180,E1 -3192.426,E2 -3192.426} C_VEL
LIN {X 0,Y 552.105,Z 365.207,A -85,B 0,C 180,E1 -3195.563,E2 -3195.563} C_VEL
LIN {X 0,Y 552.135,Z 365.21,A -85,B 0,C 180,E1 -3198.677,E2 -3198.677} C_VEL
LIN {X 0,Y 552.121,Z 365.205,A -85,B 0,C 180,E1 -3201.411,E2 -3201.411} C_VEL
LIN {X 0,Y 552.091,Z 365.214,A -85,B 0,C 180,E1 -3204.156,E2 -3204.156} C_VEL
LIN {X 0,Y 552.121,Z 365.208,A -85,B 0,C 180,E1 -3206.814,E2 -3206.814} C_VEL
LIN {X 0,Y 552.108,Z 365.206,A -85,B 0,C 180,E1 -3209.391,E2 -3209.391} C_VEL
LIN {X 0,Y 552.126,Z 365.208,A -85,B 0,C 180,E1 -3211.902,E2 -3211.902} C_VEL
LIN {X 0,Y 552.162,Z 365.203,A -85,B 0,C 180,E1 -3214.65,E2 -3214.65} C_VEL
LIN {X 0,Y 552.098,Z 365.209,A -85,B 0,C 180,E1 -3217.549,E2 -3217.549} C_VEL
LIN {X 0,Y 552.152,Z 365.207,A -85,B 0,C 180,E1 -3220.375,E2 -3220.375} C_VEL
LIN {X 0,Y 552.162,Z 365.2,A -85,B 0,C 180,E1 -3222.977,E2 -3222.977} C_VEL
LIN {X 0,Y 552.142,Z 365.211,A -85,B 0,C 180,E1 -3226.005,E2 -3226.005} C_VEL
LIN {X 0,Y 552.169,Z 365.199,A -85,B 0,C 180,E1 -3228.993,E2 -3228.993} C_VEL
LIN {X 0,Y 552.164,Z 365.209,A -85,B 0,C 180,E1 -3231.952,E2 -3231.952} C_VEL
LIN {X 0,Y 552.234,Z 365.191,A -85,B 0,C 180,E1 -3234.889,E2 -3234.889} C_VEL
LIN {X 0,Y 552.229,Z 365.2,A -85,B 0,C 180,E1 -3237.812,E2 -3237.812} C_VEL
LIN {X 0,Y 552.247,Z 365.189,A -85,B 0,C 180,E1 -3240.729,E2 -3240.729} C_VEL
LIN {X 0,Y 552.211,Z 365.194,A -85,B 0,C 180,E1 -3242.918,E2 -3242.918} C_VEL
LIN {X 0,Y 552.204,Z 365.203,A -85,B 0,C 180,E1 -3245.844,E2 -3245.844} C_VEL
LIN {X 0,Y 552.146,Z 365.202,A -85,B 0,C 180,E1 -3248.786,E2 -3248.786} C_VEL
LIN {X 0,Y 552.169,Z 365.207,A -85,B 0,C 180,E1 -3251.75,E2 -3251.75} C_VEL
LIN {X 0,Y 552.143,Z 365.202,A -85,B 0,C 180,E1 -3254.748,E2 -3254.748} C_VEL
LIN {X 0,Y 552.113,Z 365.212,A -85,B 0,C 180,E1 -3257.788,E2 -3257.788} C_VEL
LIN {X 0,Y 552.135,Z 365.205,A -85,B 0,C 180,E1 -3260.101,E2 -3260.101} C_VEL
LIN {X 0,Y 552.098,Z 365.208,A -85,B 0,C 180,E1 -3262.451,E2 -3262.451} C_VEL
LIN {X 0,Y 552.161,Z 365.209,A -85,B 0,C 180,E1 -3265.35,E2 -3265.35} C_VEL
LIN {X 0,Y 552.108,Z 365.207,A -85,B 0,C 180,E1 -3268.099,E2 -3268.099} C_VEL
LIN {X 0,Y 552.107,Z 365.207,A -85,B 0,C 180,E1 -3270.609,E2 -3270.609} C_VEL
LIN {X 0,Y 552.112,Z 365.214,A -85,B 0,C 180,E1 -3273.186,E2 -3273.186} C_VEL
LIN {X 0,Y 552.089,Z 365.21,A -85,B 0,C 180,E1 -3275.844,E2 -3275.844} C_VEL
LIN {X 0,Y 552.12,Z 365.206,A -85,B 0,C 180,E1 -3278.589,E2 -3278.589} C_VEL
LIN {X 0,Y 552.125,Z 365.209,A -85,B 0,C 180,E1 -3281.446,E2 -3281.446} C_VEL
LIN {X 0,Y 552.098,Z 365.21,A -85,B 0,C 180,E1 -3284.531,E2 -3284.531} C_VEL
LIN {X 0,Y 552.134,Z 365.206,A -85,B 0,C 180,E1 -3287.585,E2 -3287.585} C_VEL
LIN {X 0,Y 552.138,Z 365.205,A -85,B 0,C 180,E1 -3290.473,E2 -3290.473} C_VEL
LIN {X 0,Y 552.111,Z 365.21,A -85,B 0,C 180,E1 -3293.317,E2 -3293.317} C_VEL
LIN {X 0,Y 552.134,Z 365.203,A -85,B 0,C 180,E1 -3295.939,E2 -3295.939} C_VEL
LIN {X 0,Y 552.123,Z 365.209,A -85,B 0,C 180,E1 -3298.54,E2 -3298.54} C_VEL
LIN {X 0,Y 552.129,Z 365.207,A -85,B 0,C 180,E1 -3301.438,E2 -3301.438} C_VEL
LIN {X 0,Y 552.135,Z 365.209,A -85,B 0,C 180,E1 -3304.356,E2 -3304.356} C_VEL
LIN {X 0,Y 552.146,Z 365.239,A -85,B 0,C 180,E1 -3306.717,E2 -3306.717} C_VEL
LIN {X 0,Y 553.097,Z 370.546,A -85,B 0,C 180,E1 -3307.592,E2 -3307.592} C_VEL
LIN {X 0,Y 552.847,Z 387.189,A -85,B 0,C 180,E1 -3310.173,E2 -3310.173} C_VEL
LIN {X 0,Y 552.578,Z 405.623,A -85,B 0,C 180,E1 -3312.99,E2 -3312.99} C_VEL
LIN {X 0,Y 552.366,Z 422.983,A -85,B 0,C 180,E1 -3315.626,E2 -3315.626} C_VEL
LIN {X 0,Y 553.414,Z 430.791,A -85,B 0,C 180,E1 -3315.763,E2 -3315.763} C_VEL
LIN {X 0,Y 553.122,Z 530.935,A -85,B 0,C 180,E1 -3317.082,E2 -3317.082} C_VEL
LIN {X 0,Y 553.007,Z 544.21,A -85,B 0,C 180,E1 -3317.406,E2 -3317.406} C_VEL
LIN {X 0,Y 552.847,Z 556.364,A -85,B 0,C 180,E1 -3317.845,E2 -3317.845} C_VEL
LIN {X 0,Y 552.647,Z 567.248,A -85,B 0,C 180,E1 -3318.37,E2 -3318.37} C_VEL
LIN {X 0,Y 552.517,Z 578.901,A -85,B 0,C 180,E1 -3319.093,E2 -3319.093} C_VEL
LIN {X 0,Y 552.294,Z 589.535,A -85,B 0,C 180,E1 -3319.923,E2 -3319.923} C_VEL
LIN {X 0,Y 552.126,Z 599.111,A -85,B 0,C 180,E1 -3320.844,E2 -3320.844} C_VEL
LIN {X 0,Y 552.013,Z 606.959,A -85,B 0,C 180,E1 -3321.765,E2 -3321.765} C_VEL
LIN {X 0,Y 551.89,Z 614.62,A -85,B 0,C 180,E1 -3322.868,E2 -3322.868} C_VEL
LIN {X 0,Y 551.867,Z 621.679,A -85,B 0,C 180,E1 -3324.152,E2 -3324.152} C_VEL
LIN {X 0,Y 551.725,Z 626.372,A -85,B 0,C 180,E1 -3325.25,E2 -3325.25} C_VEL
LIN {X 0,Y 551.75,Z 629.958,A -85,B 0,C 180,E1 -3326.348,E2 -3326.348} C_VEL
LIN {X 0,Y 551.724,Z 631.807,A -85,B 0,C 180,E1 -3327.079,E2 -3327.079} C_VEL
LIN {X 0,Y 551.645,Z 634.183,A -85,B 0,C 180,E1 -3328.54,E2 -3328.54} C_VEL
LIN {X 0,Y 551.64,Z 635,A -85,B 0,C 180,E1 -3330,E2 -3330} C_VEL
LIN {X 0,Y 551.645,Z 634.185,A -85,B 0,C 180,E1 -3331.46,E2 -3331.46} C_VEL
LIN {X 0,Y 551.723,Z 631.81,A -85,B 0,C 180,E1 -3332.921,E2 -3332.921} C_VEL
LIN {X 0,Y 551.763,Z 628.896,A -85,B 0,C 180,E1 -3334.017,E2 -3334.017} C_VEL
LIN {X 0,Y 551.724,Z 624.949,A -85,B 0,C 180,E1 -3335.116,E2 -3335.116} C_VEL
LIN {X 0,Y 551.815,Z 619.124,A -85,B 0,C 180,E1 -3336.353,E2 -3336.353} C_VEL
LIN {X 0,Y 551.926,Z 612.237,A -85,B 0,C 180,E1 -3337.5,E2 -3337.5} C_VEL
LIN {X 0,Y 552.082,Z 603.992,A -85,B 0,C 180,E1 -3338.602,E2 -3338.602} C_VEL
LIN {X 0,Y 552.221,Z 595.54,A -85,B 0,C 180,E1 -3339.523,E2 -3339.523} C_VEL
LIN {X 0,Y 552.432,Z 585.094,A -85,B 0,C 180,E1 -3340.445,E2 -3340.445} C_VEL
LIN {X 0,Y 552.556,Z 574.288,A -85,B 0,C 180,E1 -3341.214,E2 -3341.214} C_VEL
LIN {X 0,Y 552.781,Z 563.407,A -85,B 0,C 180,E1 -3341.83,E2 -3341.83} C_VEL
LIN {X 0,Y 552.902,Z 551.765,A -85,B 0,C 180,E1 -3342.34,E2 -3342.34} C_VEL
LIN {X 0,Y 553.064,Z 539.261,A -85,B 0,C 180,E1 -3342.732,E2 -3342.732} C_VEL
LIN {X 0,Y 553.164,Z 526.603,A -85,B 0,C 180,E1 -3342.986,E2 -3342.986} C_VEL
LIN {X 0,Y 553.396,Z 429.774,A -85,B 0,C 180,E1 -3344.251,E2 -3344.251} C_VEL
LIN {X 0,Y 552.364,Z 422.884,A -85,B 0,C 180,E1 -3344.389,E2 -3344.389} C_VEL
LIN {X 0,Y 552.637,Z 402.486,A -85,B 0,C 180,E1 -3347.485,E2 -3347.485} C_VEL
LIN {X 0,Y 552.996,Z 381.846,A -85,B 0,C 180,E1 -3350.651,E2 -3350.651} C_VEL
LIN {X 0,Y 553.1,Z 370.574,A -85,B 0,C 180,E1 -3352.408,E2 -3352.408} C_VEL
LIN {X 0,Y 552.116,Z 365.215,A -85,B 0,C 180,E1 -3353.326,E2 -3353.326} C_VEL
LIN {X 0,Y 552.134,Z 365.208,A -85,B 0,C 180,E1 -3355.644,E2 -3355.644} C_VEL
LIN {X 0,Y 552.128,Z 365.207,A -85,B 0,C 180,E1 -3358.562,E2 -3358.562} C_VEL
LIN {X 0,Y 552.139,Z 365.207,A -85,B 0,C 180,E1 -3361.48,E2 -3361.48} C_VEL
LIN {X 0,Y 552.139,Z 365.203,A -85,B 0,C 180,E1 -3364.171,E2 -3364.171} C_VEL
LIN {X 0,Y 552.108,Z 365.211,A -85,B 0,C 180,E1 -3366.747,E2 -3366.747} C_VEL
LIN {X 0,Y 552.135,Z 365.205,A -85,B 0,C 180,E1 -3369.527,E2 -3369.527} C_VEL
LIN {X 0,Y 552.132,Z 365.206,A -85,B 0,C 180,E1 -3372.425,E2 -3372.425} C_VEL
LIN {X 0,Y 552.103,Z 365.208,A -85,B 0,C 180,E1 -3375.563,E2 -3375.563} C_VEL
LIN {X 0,Y 552.139,Z 365.209,A -85,B 0,C 180,E1 -3378.677,E2 -3378.677} C_VEL
LIN {X 0,Y 552.12,Z 365.207,A -85,B 0,C 180,E1 -3381.411,E2 -3381.411} C_VEL
LIN {X 0,Y 552.088,Z 365.21,A -85,B 0,C 180,E1 -3384.156,E2 -3384.156} C_VEL
LIN {X 0,Y 552.118,Z 365.214,A -85,B 0,C 180,E1 -3386.814,E2 -3386.814} C_VEL
LIN {X 0,Y 552.105,Z 365.208,A -85,B 0,C 180,E1 -3389.391,E2 -3389.391} C_VEL
LIN {X 0,Y 552.123,Z 365.205,A -85,B 0,C 180,E1 -3391.902,E2 -3391.902} C_VEL
LIN {X 0,Y 552.159,Z 365.209,A -85,B 0,C 180,E1 -3394.65,E2 -3394.65} C_VEL
LIN {X 0,Y 552.096,Z 365.208,A -85,B 0,C 180,E1 -3397.549,E2 -3397.549} C_VEL
LIN {X 0,Y 552.152,Z 365.208,A -85,B 0,C 180,E1 -3400.374,E2 -3400.374} C_VEL
LIN {X 0,Y 552.159,Z 365.203,A -85,B 0,C 180,E1 -3402.977,E2 -3402.977} C_VEL
LIN {X 0,Y 552.138,Z 365.206,A -85,B 0,C 180,E1 -3406.005,E2 -3406.005} C_VEL
LIN {X 0,Y 552.165,Z 365.201,A -85,B 0,C 180,E1 -3408.993,E2 -3408.993} C_VEL
LIN {X 0,Y 552.153,Z 365.205,A -85,B 0,C 180,E1 -3411.951,E2 -3411.951} C_VEL
LIN {X 0,Y 552.231,Z 365.193,A -85,B 0,C 180,E1 -3414.889,E2 -3414.889} C_VEL
LIN {X 0,Y 552.225,Z 365.195,A -85,B 0,C 180,E1 -3417.812,E2 -3417.812} C_VEL
LIN {X 0,Y 552.246,Z 365.191,A -85,B 0,C 180,E1 -3420.729,E2 -3420.729} C_VEL
LIN {X 0,Y 552.21,Z 365.194,A -85,B 0,C 180,E1 -3422.918,E2 -3422.918} C_VEL
LIN {X 0,Y 552.202,Z 365.2,A -85,B 0,C 180,E1 -3425.844,E2 -3425.844} C_VEL
LIN {X 0,Y 552.157,Z 365.201,A -85,B 0,C 180,E1 -3428.786,E2 -3428.786} C_VEL
LIN {X 0,Y 552.167,Z 365.204,A -85,B 0,C 180,E1 -3431.75,E2 -3431.75} C_VEL
LIN {X 0,Y 552.141,Z 365.203,A -85,B 0,C 180,E1 -3434.748,E2 -3434.748} C_VEL
LIN {X 0,Y 552.118,Z 365.213,A -85,B 0,C 180,E1 -3437.788,E2 -3437.788} C_VEL
LIN {X 0,Y 552.135,Z 365.21,A -85,B 0,C 180,E1 -3440.101,E2 -3440.101} C_VEL
LIN {X 0,Y 552.1,Z 365.209,A -85,B 0,C 180,E1 -3442.451,E2 -3442.451} C_VEL
LIN {X 0,Y 552.16,Z 365.203,A -85,B 0,C 180,E1 -3445.351,E2 -3445.351} C_VEL
LIN {X 0,Y 552.127,Z 365.209,A -85,B 0,C 180,E1 -3448.098,E2 -3448.098} C_VEL
LIN {X 0,Y 552.108,Z 365.207,A -85,B 0,C 180,E1 -3450.613,E2 -3450.613} C_VEL
LIN {X 0,Y 552.127,Z 365.207,A -85,B 0,C 180,E1 -3453.185,E2 -3453.185} C_VEL
LIN {X 0,Y 552.117,Z 365.207,A -85,B 0,C 180,E1 -3453.792,E2 -3453.792} C_VEL
LIN {X 0,Y 551.48,Z 365.289,A -85,B 0,C 180,E1 -3454.401,E2 -3454.401} C_VEL
LIN {X 0,Y 548.659,Z 365.641,A -85,B 0,C 180,E1 -3455.389,E2 -3455.389} C_VEL
LIN {X 0,Y 546.24,Z 365.94,A -85,B 0,C 180,E1 -3456.185,E2 -3456.185} C_VEL
LIN {X 0,Y 545.171,Z 366.071,A -85,B 0,C 180,E1 -3456.799,E2 -3456.799} C_VEL
LIN {X 0,Y 545.069,Z 366.085,A -85,B 0,C 180,E1 -3457.006,E2 -3457.006} C_VEL
LIN {X 0,Y 545.07,Z 366.085,A -85,B 0,C 180,E1 -3460.143,E2 -3460.143} C_VEL
LIN {X 0,Y 545.09,Z 366.084,A -85,B 0,C 180,E1 -3463.106,E2 -3463.106} C_VEL
LIN {X 0,Y 545.07,Z 366.084,A -85,B 0,C 180,E1 -3466.224,E2 -3466.224} C_VEL
LIN {X 0,Y 545.094,Z 366.082,A -85,B 0,C 180,E1 -3468.886,E2 -3468.886} C_VEL
LIN {X 0,Y 545.057,Z 366.089,A -85,B 0,C 180,E1 -3471.763,E2 -3471.763} C_VEL
LIN {X 0,Y 545.069,Z 366.084,A -85,B 0,C 180,E1 -3474.534,E2 -3474.534} C_VEL
LIN {X 0,Y 545.072,Z 366.091,A -85,B 0,C 180,E1 -3477.212,E2 -3477.212} C_VEL
LIN {X 0,Y 545.067,Z 366.086,A -85,B 0,C 180,E1 -3479.811,E2 -3479.811} C_VEL
LIN {X 0,Y 545.084,Z 366.082,A -85,B 0,C 180,E1 -3482.344,E2 -3482.344} C_VEL
LIN {X 0,Y 545.121,Z 366.082,A -85,B 0,C 180,E1 -3484.821,E2 -3484.821} C_VEL
LIN {X 0,Y 545.04,Z 366.097,A -85,B 0,C 180,E1 -3487.242,E2 -3487.242} C_VEL
LIN {X 0,Y 545.114,Z 366.205,A -85,B 0,C 180,E1 -3489.456,E2 -3489.456} C_VEL
LIN {X 0,Y 545.655,Z 369.494,A -85,B 0,C 180,E1 -3490.092,E2 -3490.092} C_VEL
LIN {X 0,Y 545.481,Z 382.312,A -85,B 0,C 180,E1 -3492.444,E2 -3492.444} C_VEL
LIN {X 0,Y 545.246,Z 398.107,A -85,B 0,C 180,E1 -3495.308,E2 -3495.308} C_VEL
LIN {X 0,Y 545.222,Z 399.122,A -85,B 0,C 180,E1 -3495.491,E2 -3495.491} C_VEL
LIN {X 0,Y 546.545,Z 407.376,A -85,B 0,C 180,E1 -3495.645,E2 -3495.645} C_VEL
LIN {X 0,Y 546.248,Z 506.057,A -85,B 0,C 180,E1 -3496.964,E2 -3496.964} C_VEL
LIN {X 0,Y 546.067,Z 519.281,A -85,B 0,C 180,E1 -3497.291,E2 -3497.291} C_VEL
LIN {X 0,Y 545.89,Z 531.414,A -85,B 0,C 180,E1 -3497.735,E2 -3497.735} C_VEL
LIN {X 0,Y 545.726,Z 543.623,A -85,B 0,C 180,E1 -3498.342,E2 -3498.342} C_VEL
LIN {X 0,Y 545.523,Z 554.577,A -85,B 0,C 180,E1 -3499.046,E2 -3499.046} C_VEL
LIN {X 0,Y 545.295,Z 565.092,A -85,B 0,C 180,E1 -3499.886,E2 -3499.886} C_VEL
LIN {X 0,Y 545.122,Z 573.686,A -85,B 0,C 180,E1 -3500.726,E2 -3500.726} C_VEL
LIN {X 0,Y 544.975,Z 581.605,A -85,B 0,C 180,E1 -3501.658,E2 -3501.658} C_VEL
LIN {X 0,Y 544.829,Z 589.353,A -85,B 0,C 180,E1 -3502.775,E2 -3502.775} C_VEL
LIN {X 0,Y 544.778,Z 596.46,A -85,B 0,C 180,E1 -3504.076,E2 -3504.076} C_VEL
LIN {X 0,Y 544.629,Z 601.2,A -85,B 0,C 180,E1 -3505.189,E2 -3505.189} C_VEL
LIN {X 0,Y 544.669,Z 604.831,A -85,B 0,C 180,E1 -3506.301,E2 -3506.301} C_VEL
LIN {X 0,Y 544.65,Z 606.708,A -85,B 0,C 180,E1 -3507.041,E2 -3507.041} C_VEL
LIN {X 0,Y 544.571,Z 608.128,A -85,B 0,C 180,E1 -3507.781,E2 -3507.781} C_VEL
LIN {X 0,Y 544.542,Z 609.757,A -85,B 0,C 180,E1 -3509.261,E2 -3509.261} C_VEL
LIN {X 0,Y 544.542,Z 609.996,A -85,B 0,C 180,E1 -3510,E2 -3510} C_VEL
LIN {X 0,Y 544.542,Z 609.814,A -85,B 0,C 180,E1 -3510.74,E2 -3510.74} C_VEL
LIN {X 0,Y 544.572,Z 608.262,A -85,B 0,C 180,E1 -3512.219,E2 -3512.219} C_VEL
LIN {X 0,Y 544.651,Z 606.901,A -85,B 0,C 180,E1 -3512.959,E2 -3512.959} C_VEL
LIN {X 0,Y 544.684,Z 604.023,A -85,B 0,C 180,E1 -3514.07,E2 -3514.07} C_VEL
LIN {X 0,Y 544.653,Z 600.121,A -85,B 0,C 180,E1 -3515.182,E2 -3515.182} C_VEL
LIN {X 0,Y 544.725,Z 594.897,A -85,B 0,C 180,E1 -3516.335,E2 -3516.335} C_VEL
LIN {X 0,Y 544.859,Z 587.531,A -85,B 0,C 180,E1 -3517.598,E2 -3517.598} C_VEL
LIN {X 0,Y 544.999,Z 579.348,A -85,B 0,C 180,E1 -3518.715,E2 -3518.715} C_VEL
LIN {X 0,Y 545.159,Z 570.978,A -85,B 0,C 180,E1 -3519.648,E2 -3519.648} C_VEL
LIN {X 0,Y 545.383,Z 560.651,A -85,B 0,C 180,E1 -3520.582,E2 -3520.582} C_VEL
LIN {X 0,Y 545.601,Z 549.249,A -85,B 0,C 180,E1 -3521.406,E2 -3521.406} C_VEL
LIN {X 0,Y 545.808,Z 537.431,A -85,B 0,C 180,E1 -3522.078,E2 -3522.078} C_VEL
LIN {X 0,Y 545.991,Z 525.406,A -85,B 0,C 180,E1 -3522.593,E2 -3522.593} C_VEL
LIN {X 0,Y 546.158,Z 512.338,A -85,B 0,C 180,E1 -3522.991,E2 -3522.991} C_VEL
LIN {X 0,Y 546.291,Z 499.903,A -85,B 0,C 180,E1 -3523.224,E2 -3523.224} C_VEL
LIN {X 0,Y 546.446,Z 406.292,A -85,B 0,C 180,E1 -3524.462,E2 -3524.462} C_VEL
LIN {X 0,Y 545.215,Z 399.16,A -85,B 0,C 180,E1 -3524.594,E2 -3524.594} C_VEL
LIN {X 0,Y 545.457,Z 384.548,A -85,B 0,C 180,E1 -3527.239,E2 -3527.239} C_VEL
LIN {X 0,Y 545.662,Z 371.844,A -85,B 0,C 180,E1 -3529.565,E2 -3529.565} C_VEL
LIN {X 0,Y 545.388,Z 367.614,A -85,B 0,C 180,E1 -3530.361,E2 -3530.361} C_VEL
LIN {X 0,Y 545.124,Z 366.086,A -85,B 0,C 180,E1 -3530.667,E2 -3530.667} C_VEL
LIN {X 0,Y 545.059,Z 366.088,A -85,B 0,C 180,E1 -3533.726,E2 -3533.726} C_VEL
LIN {X 0,Y 545.084,Z 366.085,A -85,B 0,C 180,E1 -3536.001,E2 -3536.001} C_VEL
LIN {X 0,Y 545.094,Z 366.089,A -85,B 0,C 180,E1 -3538.748,E2 -3538.748} C_VEL
LIN {X 0,Y 545.062,Z 366.084,A -85,B 0,C 180,E1 -3541.679,E2 -3541.679} C_VEL
LIN {X 0,Y 545.078,Z 366.089,A -85,B 0,C 180,E1 -3544.564,E2 -3544.564} C_VEL
LIN {X 0,Y 545.04,Z 366.088,A -85,B 0,C 180,E1 -3547.304,E2 -3547.304} C_VEL
LIN {X 0,Y 545.07,Z 366.086,A -85,B 0,C 180,E1 -3550.143,E2 -3550.143} C_VEL
LIN {X 0,Y 545.083,Z 366.084,A -85,B 0,C 180,E1 -3553.107,E2 -3553.107} C_VEL
LIN {X 0,Y 545.07,Z 366.088,A -85,B 0,C 180,E1 -3556.225,E2 -3556.225} C_VEL
LIN {X 0,Y 545.093,Z 366.084,A -85,B 0,C 180,E1 -3558.886,E2 -3558.886} C_VEL
LIN {X 0,Y 545.056,Z 366.086,A -85,B 0,C 180,E1 -3561.763,E2 -3561.763} C_VEL
LIN {X 0,Y 545.042,Z 366.094,A -85,B 0,C 180,E1 -3564.532,E2 -3564.532} C_VEL
LIN {X 0,Y 545.074,Z 366.083,A -85,B 0,C 180,E1 -3567.212,E2 -3567.212} C_VEL
LIN {X 0,Y 545.069,Z 366.086,A -85,B 0,C 180,E1 -3569.811,E2 -3569.811} C_VEL
LIN {X 0,Y 545.095,Z 366.089,A -85,B 0,C 180,E1 -3572.344,E2 -3572.344} C_VEL
LIN {X 0,Y 545.123,Z 366.078,A -85,B 0,C 180,E1 -3574.821,E2 -3574.821} C_VEL
LIN {X 0,Y 545.043,Z 366.087,A -85,B 0,C 180,E1 -3577.242,E2 -3577.242} C_VEL
LIN {X 0,Y 545.124,Z 366.082,A -85,B 0,C 180,E1 -3580.415,E2 -3580.415} C_VEL
LIN {X 0,Y 545.077,Z 366.084,A -85,B 0,C 180,E1 -3583.521,E2 -3583.521} C_VEL
LIN {X 0,Y 545.101,Z 366.085,A -85,B 0,C 180,E1 -3585.82,E2 -3585.82} C_VEL
LIN {X 0,Y 545.124,Z 366.077,A -85,B 0,C 180,E1 -3588.849,E2 -3588.849} C_VEL
LIN {X 0,Y 545.134,Z 366.083,A -85,B 0,C 180,E1 -3591.847,E2 -3591.847} C_VEL
LIN {X 0,Y 545.209,Z 366.066,A -85,B 0,C 180,E1 -3594.823,E2 -3594.823} C_VEL
LIN {X 0,Y 545.201,Z 366.075,A -85,B 0,C 180,E1 -3597.784,E2 -3597.784} C_VEL
LIN {X 0,Y 545.217,Z 366.065,A -85,B 0,C 180,E1 -3600.739,E2 -3600.739} C_VEL
LIN {X 0,Y 545.178,Z 366.07,A -85,B 0,C 180,E1 -3602.956,E2 -3602.956} C_VEL
LIN {X 0,Y 545.176,Z 366.077,A -85,B 0,C 180,E1 -3605.919,E2 -3605.919} C_VEL
LIN {X 0,Y 545.107,Z 366.079,A -85,B 0,C 180,E1 -3608.9,E2 -3608.9} C_VEL
LIN {X 0,Y 545.141,Z 366.08,A -85,B 0,C 180,E1 -3611.904,E2 -3611.904} C_VEL
LIN {X 0,Y 545.092,Z 366.082,A -85,B 0,C 180,E1 -3614.943,E2 -3614.943} C_VEL
LIN {X 0,Y 545.081,Z 366.085,A -85,B 0,C 180,E1 -3618.026,E2 -3618.026} C_VEL
LIN {X 0,Y 545.1,Z 366.08,A -85,B 0,C 180,E1 -3620.372,E2 -3620.372} C_VEL
LIN {X 0,Y 545.085,Z 366.089,A -85,B 0,C 180,E1 -3623.559,E2 -3623.559} C_VEL
LIN {X 0,Y 545.082,Z 366.083,A -85,B 0,C 180,E1 -3626,E2 -3626} C_VEL
LIN {X 0,Y 545.094,Z 366.082,A -85,B 0,C 180,E1 -3628.748,E2 -3628.748} C_VEL
LIN {X 0,Y 545.062,Z 366.088,A -85,B 0,C 180,E1 -3631.679,E2 -3631.679} C_VEL
LIN {X 0,Y 545.062,Z 366.085,A -85,B 0,C 180,E1 -3634.565,E2 -3634.565} C_VEL
LIN {X 0,Y 545.041,Z 366.095,A -85,B 0,C 180,E1 -3637.304,E2 -3637.304} C_VEL
LIN {X 0,Y 545.069,Z 366.083,A -85,B 0,C 180,E1 -3640.143,E2 -3640.143} C_VEL
LIN {X 0,Y 545.083,Z 366.091,A -85,B 0,C 180,E1 -3643.106,E2 -3643.106} C_VEL
LIN {X 0,Y 545.053,Z 366.085,A -85,B 0,C 180,E1 -3646.226,E2 -3646.226} C_VEL
LIN {X 0,Y 545.085,Z 366.088,A -85,B 0,C 180,E1 -3648.885,E2 -3648.885} C_VEL
LIN {X 0,Y 545.088,Z 366.087,A -85,B 0,C 180,E1 -3650.819,E2 -3650.819} C_VEL
LIN {X 0,Y 545.047,Z 366.087,A -85,B 0,C 180,E1 -3653.62,E2 -3653.62} C_VEL
LIN {X 0,Y 545.072,Z 366.085,A -85,B 0,C 180,E1 -3656.328,E2 -3656.328} C_VEL
LIN {X 0,Y 545.072,Z 366.092,A -85,B 0,C 180,E1 -3658.952,E2 -3658.952} C_VEL
LIN {X 0,Y 545.106,Z 366.082,A -85,B 0,C 180,E1 -3661.508,E2 -3661.508} C_VEL
LIN {X 0,Y 545.1,Z 366.087,A -85,B 0,C 180,E1 -3664.491,E2 -3664.491} C_VEL
LIN {X 0,Y 545.093,Z 366.151,A -85,B 0,C 180,E1 -3666.567,E2 -3666.567} C_VEL
LIN {X 0,Y 546.187,Z 372.661,A -85,B 0,C 180,E1 -3667.651,E2 -3667.651} C_VEL
LIN {X 0,Y 545.888,Z 388.537,A -85,B 0,C 180,E1 -3670.142,E2 -3670.142} C_VEL
LIN {X 0,Y 545.562,Z 406.728,A -85,B 0,C 180,E1 -3672.958,E2 -3672.958} C_VEL
LIN {X 0,Y 545.36,Z 422.96,A -85,B 0,C 180,E1 -3675.44,E2 -3675.44} C_VEL
LIN {X 0,Y 546.553,Z 431.857,A -85,B 0,C 180,E1 -3675.594,E2 -3675.594} C_VEL
LIN {X 0,Y 546.202,Z 530.935,A -85,B 0,C 180,E1 -3676.916,E2 -3676.916} C_VEL
LIN {X 0,Y 546.082,Z 544.209,A -85,B 0,C 180,E1 -3677.244,E2 -3677.244} C_VEL
LIN {X 0,Y 545.894,Z 556.363,A -85,B 0,C 180,E1 -3677.688,E2 -3677.688} C_VEL
LIN {X 0,Y 545.679,Z 567.461,A -85,B 0,C 180,E1 -3678.23,E2 -3678.23} C_VEL
LIN {X 0,Y 545.521,Z 578.899,A -85,B 0,C 180,E1 -3678.952,E2 -3678.952} C_VEL
LIN {X 0,Y 545.286,Z 589.534,A -85,B 0,C 180,E1 -3679.792,E2 -3679.792} C_VEL
LIN {X 0,Y 545.084,Z 599.111,A -85,B 0,C 180,E1 -3680.725,E2 -3680.725} C_VEL
LIN {X 0,Y 544.978,Z 606.959,A -85,B 0,C 180,E1 -3681.658,E2 -3681.658} C_VEL
LIN {X 0,Y 544.824,Z 614.62,A -85,B 0,C 180,E1 -3682.775,E2 -3682.775} C_VEL
LIN {X 0,Y 544.776,Z 621.679,A -85,B 0,C 180,E1 -3684.076,E2 -3684.076} C_VEL
LIN {X 0,Y 544.629,Z 626.372,A -85,B 0,C 180,E1 -3685.188,E2 -3685.188} C_VEL
LIN {X 0,Y 544.669,Z 629.958,A -85,B 0,C 180,E1 -3686.301,E2 -3686.301} C_VEL
LIN {X 0,Y 544.65,Z 631.807,A -85,B 0,C 180,E1 -3687.041,E2 -3687.041} C_VEL
LIN {X 0,Y 544.546,Z 634.183,A -85,B 0,C 180,E1 -3688.521,E2 -3688.521} C_VEL
LIN {X 0,Y 544.541,Z 635,A -85,B 0,C 180,E1 -3690,E2 -3690} C_VEL
LIN {X 0,Y 544.546,Z 634.184,A -85,B 0,C 180,E1 -3691.479,E2 -3691.479} C_VEL
LIN {X 0,Y 544.65,Z 631.81,A -85,B 0,C 180,E1 -3692.959,E2 -3692.959} C_VEL
LIN {X 0,Y 544.683,Z 628.896,A -85,B 0,C 180,E1 -3694.069,E2 -3694.069} C_VEL
LIN {X 0,Y 544.654,Z 624.949,A -85,B 0,C 180,E1 -3695.182,E2 -3695.182} C_VEL
LIN {X 0,Y 544.73,Z 619.643,A -85,B 0,C 180,E1 -3696.34,E2 -3696.34} C_VEL
LIN {X 0,Y 544.836,Z 613.467,A -85,B 0,C 180,E1 -3697.411,E2 -3697.411} C_VEL
LIN {X 0,Y 545.006,Z 605.478,A -85,B 0,C 180,E1 -3698.528,E2 -3698.528} C_VEL
LIN {X 0,Y 545.152,Z 597.334,A -85,B 0,C 180,E1 -3699.461,E2 -3699.461} C_VEL
LIN {X 0,Y 545.376,Z 587.398,A -85,B 0,C 180,E1 -3700.394,E2 -3700.394} C_VEL
LIN {X 0,Y 545.57,Z 576.593,A -85,B 0,C 180,E1 -3701.208,E2 -3701.208} C_VEL
LIN {X 0,Y 545.747,Z 565.172,A -85,B 0,C 180,E1 -3701.891,E2 -3701.891} C_VEL
LIN {X 0,Y 545.937,Z 552.973,A -85,B 0,C 180,E1 -3702.452,E2 -3702.452} C_VEL
LIN {X 0,Y 546.148,Z 540.175,A -85,B 0,C 180,E1 -3702.872,E2 -3702.872} C_VEL
LIN {X 0,Y 546.252,Z 526.602,A -85,B 0,C 180,E1 -3703.154,E2 -3703.154} C_VEL
LIN {X 0,Y 546.427,Z 429.804,A -85,B 0,C 180,E1 -3704.436,E2 -3704.436} C_VEL
LIN {X 0,Y 545.342,Z 422.842,A -85,B 0,C 180,E1 -3704.578,E2 -3704.578} C_VEL
LIN {X 0,Y 545.662,Z 402.138,A -85,B 0,C 180,E1 -3707.747,E2 -3707.747} C_VEL
LIN {X 0,Y 546.032,Z 382.954,A -85,B 0,C 180,E1 -3710.729,E2 -3710.729} C_VEL
LIN {X 0,Y 546.124,Z 371.543,A -85,B 0,C 180,E1 -3712.532,E2 -3712.532} C_VEL
LIN {X 0,Y 545.096,Z 366.09,A -85,B 0,C 180,E1 -3713.458,E2 -3713.458} C_VEL
LIN {X 0,Y 545.083,Z 366.083,A -85,B 0,C 180,E1 -3716,E2 -3716} C_VEL
LIN {X 0,Y 545.092,Z 366.086,A -85,B 0,C 180,E1 -3718.748,E2 -3718.748} C_VEL
LIN {X 0,Y 545.081,Z 366.084,A -85,B 0,C 180,E1 -3721.682,E2 -3721.682} C_VEL
LIN {X 0,Y 545.079,Z 366.084,A -85,B 0,C 180,E1 -3724.563,E2 -3724.563} C_VEL
LIN {X 0,Y 545.04,Z 366.092,A -85,B 0,C 180,E1 -3727.304,E2 -3727.304} C_VEL
LIN {X 0,Y 545.074,Z 366.083,A -85,B 0,C 180,E1 -3730.142,E2 -3730.142} C_VEL
LIN {X 0,Y 545.081,Z 366.089,A -85,B 0,C 180,E1 -3733.107,E2 -3733.107} C_VEL
LIN {X 0,Y 545.068,Z 366.085,A -85,B 0,C 180,E1 -3736.224,E2 -3736.224} C_VEL
LIN {X 0,Y 545.095,Z 366.089,A -85,B 0,C 180,E1 -3738.886,E2 -3738.886} C_VEL
LIN {X 0,Y 545.054,Z 366.085,A -85,B 0,C 180,E1 -3741.763,E2 -3741.763} C_VEL
LIN {X 0,Y 545.039,Z 366.093,A -85,B 0,C 180,E1 -3744.532,E2 -3744.532} C_VEL
LIN {X 0,Y 545.072,Z 366.086,A -85,B 0,C 180,E1 -3747.212,E2 -3747.212} C_VEL
LIN {X 0,Y 545.066,Z 366.084,A -85,B 0,C 180,E1 -3749.811,E2 -3749.811} C_VEL
LIN {X 0,Y 545.092,Z 366.085,A -85,B 0,C 180,E1 -3752.344,E2 -3752.344} C_VEL
LIN {X 0,Y 545.12,Z 366.083,A -85,B 0,C 180,E1 -3754.82,E2 -3754.82} C_VEL
LIN {X 0,Y 545.041,Z 366.088,A -85,B 0,C 180,E1 -3757.242,E2 -3757.242} C_VEL
LIN {X 0,Y 545.124,Z 366.085,A -85,B 0,C 180,E1 -3760.415,E2 -3760.415} C_VEL
LIN {X 0,Y 545.076,Z 366.082,A -85,B 0,C 180,E1 -3763.521,E2 -3763.521} C_VEL
LIN {X 0,Y 545.098,Z 366.081,A -85,B 0,C 180,E1 -3765.82,E2 -3765.82} C_VEL
LIN {X 0,Y 545.121,Z 366.08,A -85,B 0,C 180,E1 -3768.849,E2 -3768.849} C_VEL
LIN {X 0,Y 545.102,Z 366.082,A -85,B 0,C 180,E1 -3771.847,E2 -3771.847} C_VEL
LIN {X 0,Y 545.207,Z 366.068,A -85,B 0,C 180,E1 -3774.823,E2 -3774.823} C_VEL
LIN {X 0,Y 545.197,Z 366.07,A -85,B 0,C 180,E1 -3777.784,E2 -3777.784} C_VEL
LIN {X 0,Y 545.216,Z 366.067,A -85,B 0,C 180,E1 -3780.739,E2 -3780.739} C_VEL
LIN {X 0,Y 545.176,Z 366.07,A -85,B 0,C 180,E1 -3782.956,E2 -3782.956} C_VEL
LIN {X 0,Y 545.174,Z 366.077,A -85,B 0,C 180,E1 -3785.92,E2 -3785.92} C_VEL
LIN {X 0,Y 545.115,Z 366.078,A -85,B 0,C 180,E1 -3788.9,E2 -3788.9} C_VEL
LIN {X 0,Y 545.139,Z 366.082,A -85,B 0,C 180,E1 -3791.904,E2 -3791.904} C_VEL
LIN {X 0,Y 545.09,Z 366.081,A -85,B 0,C 180,E1 -3794.944,E2 -3794.944} C_VEL
LIN {X 0,Y 545.086,Z 366.089,A -85,B 0,C 180,E1 -3798.026,E2 -3798.026} C_VEL
LIN {X 0,Y 545.099,Z 366.082,A -85,B 0,C 180,E1 -3800.372,E2 -3800.372} C_VEL
LIN {X 0,Y 545.096,Z 366.085,A -85,B 0,C 180,E1 -3803.559,E2 -3803.559} C_VEL
LIN {X 0,Y 545.084,Z 366.088,A -85,B 0,C 180,E1 -3806,E2 -3806} C_VEL
LIN {X 0,Y 545.093,Z 366.08,A -85,B 0,C 180,E1 -3808.748,E2 -3808.748} C_VEL
LIN {X 0,Y 545.063,Z 366.093,A -85,B 0,C 180,E1 -3811.679,E2 -3811.679} C_VEL
LIN {X 0,Y 545.08,Z 366.082,A -85,B 0,C 180,E1 -3814.563,E2 -3814.563} C_VEL
LIN {X 0,Y 545.069,Z 366.085,A -85,B 0,C 180,E1 -3817.006,E2 -3817.006} C_VEL
LIN {X 0,Y 544.36,Z 366.182,A -85,B 0,C 180,E1 -3817.623,E2 -3817.623} C_VEL
LIN {X 0,Y 541.493,Z 366.537,A -85,B 0,C 180,E1 -3818.624,E2 -3818.624} C_VEL
LIN {X 0,Y 539.106,Z 366.833,A -85,B 0,C 180,E1 -3819.43,E2 -3819.43} C_VEL
LIN {X 0,Y 538.096,Z 366.955,A -85,B 0,C 180,E1 -3820.052,E2 -3820.052} C_VEL
LIN {X 0,Y 538.021,Z 366.962,A -85,B 0,C 180,E1 -3820.262,E2 -3820.262} C_VEL
LIN {X 0,Y 538.037,Z 366.961,A -85,B 0,C 180,E1 -3822.988,E2 -3822.988} C_VEL
LIN {X 0,Y 538.033,Z 366.963,A -85,B 0,C 180,E1 -3825.925,E2 -3825.925} C_VEL
LIN {X 0,Y 538.054,Z 366.964,A -85,B 0,C 180,E1 -3829.252,E2 -3829.252} C_VEL
LIN {X 0,Y 537.997,Z 366.965,A -85,B 0,C 180,E1 -3832.123,E2 -3832.123} C_VEL
LIN {X 0,Y 538.024,Z 366.964,A -85,B 0,C 180,E1 -3834.917,E2 -3834.917} C_VEL
LIN {X 0,Y 538.022,Z 366.966,A -85,B 0,C 180,E1 -3837.617,E2 -3837.617} C_VEL
LIN {X 0,Y 538.021,Z 366.961,A -85,B 0,C 180,E1 -3840.239,E2 -3840.239} C_VEL
LIN {X 0,Y 538.06,Z 366.96,A -85,B 0,C 180,E1 -3842.796,E2 -3842.796} C_VEL
LIN {X 0,Y 538.051,Z 366.966,A -85,B 0,C 180,E1 -3845.293,E2 -3845.293} C_VEL
LIN {X 0,Y 538.028,Z 366.966,A -85,B 0,C 180,E1 -3848.546,E2 -3848.546} C_VEL
LIN {X 0,Y 538.081,Z 367.007,A -85,B 0,C 180,E1 -3849.3,E2 -3849.3} C_VEL
LIN {X 0,Y 538.691,Z 371.489,A -85,B 0,C 180,E1 -3850.171,E2 -3850.171} C_VEL
LIN {X 0,Y 538.491,Z 384.198,A -85,B 0,C 180,E1 -3852.532,E2 -3852.532} C_VEL
LIN {X 0,Y 538.248,Z 399.511,A -85,B 0,C 180,E1 -3855.309,E2 -3855.309} C_VEL
LIN {X 0,Y 539.695,Z 409.134,A -85,B 0,C 180,E1 -3855.48,E2 -3855.48} C_VEL
LIN {X 0,Y 539.36,Z 506.249,A -85,B 0,C 180,E1 -3856.795,E2 -3856.795} C_VEL
LIN {X 0,Y 539.156,Z 519.452,A -85,B 0,C 180,E1 -3857.125,E2 -3857.125} C_VEL
LIN {X 0,Y 538.974,Z 531.562,A -85,B 0,C 180,E1 -3857.576,E2 -3857.576} C_VEL
LIN {X 0,Y 538.771,Z 543.744,A -85,B 0,C 180,E1 -3858.19,E2 -3858.19} C_VEL
LIN {X 0,Y 538.511,Z 555.957,A -85,B 0,C 180,E1 -3858.997,E2 -3858.997} C_VEL
LIN {X 0,Y 538.28,Z 566.217,A -85,B 0,C 180,E1 -3859.848,E2 -3859.848} C_VEL
LIN {X 0,Y 538.081,Z 575.424,A -85,B 0,C 180,E1 -3860.793,E2 -3860.793} C_VEL
LIN {X 0,Y 537.862,Z 584.366,A -85,B 0,C 180,E1 -3861.925,E2 -3861.925} C_VEL
LIN {X 0,Y 537.741,Z 591.587,A -85,B 0,C 180,E1 -3863.056,E2 -3863.056} C_VEL
LIN {X 0,Y 537.694,Z 596.463,A -85,B 0,C 180,E1 -3863.998,E2 -3863.998} C_VEL
LIN {X 0,Y 537.541,Z 601.202,A -85,B 0,C 180,E1 -3865.125,E2 -3865.125} C_VEL
LIN {X 0,Y 537.591,Z 604.833,A -85,B 0,C 180,E1 -3866.252,E2 -3866.252} C_VEL
LIN {X 0,Y 537.551,Z 606.71,A -85,B 0,C 180,E1 -3867.002,E2 -3867.002} C_VEL
LIN {X 0,Y 537.49,Z 608.129,A -85,B 0,C 180,E1 -3867.752,E2 -3867.752} C_VEL
LIN {X 0,Y 537.442,Z 609.757,A -85,B 0,C 180,E1 -3869.251,E2 -3869.251} C_VEL
LIN {X 0,Y 537.442,Z 609.996,A -85,B 0,C 180,E1 -3870,E2 -3870} C_VEL
LIN {X 0,Y 537.442,Z 609.814,A -85,B 0,C 180,E1 -3870.749,E2 -3870.749} C_VEL
LIN {X 0,Y 537.49,Z 608.26,A -85,B 0,C 180,E1 -3872.248,E2 -3872.248} C_VEL
LIN {X 0,Y 537.552,Z 606.899,A -85,B 0,C 180,E1 -3872.998,E2 -3872.998} C_VEL
LIN {X 0,Y 537.604,Z 604.021,A -85,B 0,C 180,E1 -3874.123,E2 -3874.123} C_VEL
LIN {X 0,Y 537.587,Z 600.119,A -85,B 0,C 180,E1 -3875.251,E2 -3875.251} C_VEL
LIN {X 0,Y 537.639,Z 595.367,A -85,B 0,C 180,E1 -3876.321,E2 -3876.321} C_VEL
LIN {X 0,Y 537.79,Z 588.755,A -85,B 0,C 180,E1 -3877.509,E2 -3877.509} C_VEL
LIN {X 0,Y 537.952,Z 580.833,A -85,B 0,C 180,E1 -3878.641,E2 -3878.641} C_VEL
LIN {X 0,Y 538.132,Z 571.011,A -85,B 0,C 180,E1 -3879.775,E2 -3879.775} C_VEL
LIN {X 0,Y 538.375,Z 560.713,A -85,B 0,C 180,E1 -3880.721,E2 -3880.721} C_VEL
LIN {X 0,Y 538.624,Z 549.717,A -85,B 0,C 180,E1 -3881.531,E2 -3881.531} C_VEL
LIN {X 0,Y 538.842,Z 539.353,A -85,B 0,C 180,E1 -3882.141,E2 -3882.141} C_VEL
LIN {X 0,Y 539.012,Z 528.048,A -85,B 0,C 180,E1 -3882.663,E2 -3882.663} C_VEL
LIN {X 0,Y 539.251,Z 515.216,A -85,B 0,C 180,E1 -3883.088,E2 -3883.088} C_VEL
LIN {X 0,Y 539.371,Z 501.565,A -85,B 0,C 180,E1 -3883.373,E2 -3883.373} C_VEL
LIN {X 0,Y 539.569,Z 407.255,A -85,B 0,C 180,E1 -3884.639,E2 -3884.639} C_VEL
LIN {X 0,Y 538.231,Z 399.281,A -85,B 0,C 180,E1 -3884.793,E2 -3884.793} C_VEL
LIN {X 0,Y 538.502,Z 383.502,A -85,B 0,C 180,E1 -3887.687,E2 -3887.687} C_VEL
LIN {X 0,Y 538.688,Z 370.759,A -85,B 0,C 180,E1 -3890.057,E2 -3890.057} C_VEL
LIN {X 0,Y 538.047,Z 366.968,A -85,B 0,C 180,E1 -3890.801,E2 -3890.801} C_VEL
LIN {X 0,Y 538.007,Z 366.967,A -85,B 0,C 180,E1 -3893.889,E2 -3893.889} C_VEL
LIN {X 0,Y 538.046,Z 366.964,A -85,B 0,C 180,E1 -3896.367,E2 -3896.367} C_VEL
LIN {X 0,Y 538.035,Z 366.967,A -85,B 0,C 180,E1 -3898.934,E2 -3898.934} C_VEL
LIN {X 0,Y 538.014,Z 366.962,A -85,B 0,C 180,E1 -3901.887,E2 -3901.887} C_VEL
LIN {X 0,Y 538.027,Z 366.968,A -85,B 0,C 180,E1 -3904.619,E2 -3904.619} C_VEL
LIN {X 0,Y 538.009,Z 366.966,A -85,B 0,C 180,E1 -3907.17,E2 -3907.17} C_VEL
LIN {X 0,Y 538.027,Z 366.961,A -85,B 0,C 180,E1 -3909.797,E2 -3909.797} C_VEL
LIN {X 0,Y 538.023,Z 366.967,A -85,B 0,C 180,E1 -3912.786,E2 -3912.786} C_VEL
LIN {X 0,Y 538.034,Z 366.961,A -85,B 0,C 180,E1 -3915.926,E2 -3915.926} C_VEL
LIN {X 0,Y 538.054,Z 366.958,A -85,B 0,C 180,E1 -3919.224,E2 -3919.224} C_VEL
LIN {X 0,Y 537.996,Z 366.969,A -85,B 0,C 180,E1 -3922.122,E2 -3922.122} C_VEL
LIN {X 0,Y 538.004,Z 366.966,A -85,B 0,C 180,E1 -3924.916,E2 -3924.916} C_VEL
LIN {X 0,Y 538.024,Z 366.962,A -85,B 0,C 180,E1 -3927.617,E2 -3927.617} C_VEL
LIN {X 0,Y 538.023,Z 366.97,A -85,B 0,C 180,E1 -3930.239,E2 -3930.239} C_VEL
LIN {X 0,Y 538.069,Z 366.958,A -85,B 0,C 180,E1 -3932.796,E2 -3932.796} C_VEL
LIN {X 0,Y 538.033,Z 366.96,A -85,B 0,C 180,E1 -3935.292,E2 -3935.292} C_VEL
LIN {X 0,Y 538.021,Z 366.969,A -85,B 0,C 180,E1 -3938.042,E2 -3938.042} C_VEL
LIN {X 0,Y 538.042,Z 366.959,A -85,B 0,C 180,E1 -3940.94,E2 -3940.94} C_VEL
LIN {X 0,Y 538.029,Z 366.961,A -85,B 0,C 180,E1 -3943.299,E2 -3943.299} C_VEL
LIN {X 0,Y 538.07,Z 366.958,A -85,B 0,C 180,E1 -3945.631,E2 -3945.631} C_VEL
LIN {X 0,Y 538.084,Z 366.954,A -85,B 0,C 180,E1 -3948.702,E2 -3948.702} C_VEL
LIN {X 0,Y 538.09,Z 366.959,A -85,B 0,C 180,E1 -3951.74,E2 -3951.74} C_VEL
LIN {X 0,Y 538.167,Z 366.943,A -85,B 0,C 180,E1 -3954.755,E2 -3954.755} C_VEL
LIN {X 0,Y 538.173,Z 366.95,A -85,B 0,C 180,E1 -3957.755,E2 -3957.755} C_VEL
LIN {X 0,Y 538.188,Z 366.941,A -85,B 0,C 180,E1 -3960.748,E2 -3960.748} C_VEL
LIN {X 0,Y 538.144,Z 366.946,A -85,B 0,C 180,E1 -3962.994,E2 -3962.994} C_VEL
LIN {X 0,Y 538.129,Z 366.953,A -85,B 0,C 180,E1 -3965.997,E2 -3965.997} C_VEL
LIN {X 0,Y 538.059,Z 366.958,A -85,B 0,C 180,E1 -3969.018,E2 -3969.018} C_VEL
LIN {X 0,Y 538.089,Z 366.956,A -85,B 0,C 180,E1 -3972.062,E2 -3972.062} C_VEL
LIN {X 0,Y 538.051,Z 366.961,A -85,B 0,C 180,E1 -3975.144,E2 -3975.144} C_VEL
LIN {X 0,Y 538.033,Z 366.961,A -85,B 0,C 180,E1 -3978.27,E2 -3978.27} C_VEL
LIN {X 0,Y 538.045,Z 366.959,A -85,B 0,C 180,E1 -3980.651,E2 -3980.651} C_VEL
LIN {X 0,Y 538.008,Z 366.966,A -85,B 0,C 180,E1 -3983.888,E2 -3983.888} C_VEL
LIN {X 0,Y 538.044,Z 366.958,A -85,B 0,C 180,E1 -3986.367,E2 -3986.367} C_VEL
LIN {X 0,Y 538.035,Z 366.963,A -85,B 0,C 180,E1 -3988.933,E2 -3988.933} C_VEL
LIN {X 0,Y 538.015,Z 366.964,A -85,B 0,C 180,E1 -3991.887,E2 -3991.887} C_VEL
LIN {X 0,Y 538.013,Z 366.964,A -85,B 0,C 180,E1 -3994.617,E2 -3994.617} C_VEL
LIN {X 0,Y 538.009,Z 366.972,A -85,B 0,C 180,E1 -3997.17,E2 -3997.17} C_VEL
LIN {X 0,Y 538.026,Z 366.962,A -85,B 0,C 180,E1 -3999.797,E2 -3999.797} C_VEL
LIN {X 0,Y 538.023,Z 366.965,A -85,B 0,C 180,E1 -4002.786,E2 -4002.786} C_VEL
LIN {X 0,Y 538.033,Z 366.969,A -85,B 0,C 180,E1 -4005.14,E2 -4005.14} C_VEL
LIN {X 0,Y 538.034,Z 366.96,A -85,B 0,C 180,E1 -4008.227,E2 -4008.227} C_VEL
LIN {X 0,Y 538.02,Z 366.968,A -85,B 0,C 180,E1 -4011.17,E2 -4011.17} C_VEL
LIN {X 0,Y 538.001,Z 366.964,A -85,B 0,C 180,E1 -4014.088,E2 -4014.088} C_VEL
LIN {X 0,Y 538.034,Z 366.966,A -85,B 0,C 180,E1 -4016.727,E2 -4016.727} C_VEL
LIN {X 0,Y 538.031,Z 366.963,A -85,B 0,C 180,E1 -4019.556,E2 -4019.556} C_VEL
LIN {X 0,Y 538.044,Z 366.961,A -85,B 0,C 180,E1 -4021.95,E2 -4021.95} C_VEL
LIN {X 0,Y 538.076,Z 366.962,A -85,B 0,C 180,E1 -4024.467,E2 -4024.467} C_VEL
LIN {X 0,Y 538.073,Z 367.119,A -85,B 0,C 180,E1 -4026.423,E2 -4026.423} C_VEL
LIN {X 0,Y 539.205,Z 373.033,A -85,B 0,C 180,E1 -4027.427,E2 -4027.427} C_VEL
LIN {X 0,Y 538.931,Z 388.377,A -85,B 0,C 180,E1 -4029.872,E2 -4029.872} C_VEL
LIN {X 0,Y 538.6,Z 406.581,A -85,B 0,C 180,E1 -4032.731,E2 -4032.731} C_VEL
LIN {X 0,Y 538.339,Z 422.834,A -85,B 0,C 180,E1 -4035.249,E2 -4035.249} C_VEL
LIN {X 0,Y 539.687,Z 431.956,A -85,B 0,C 180,E1 -4035.411,E2 -4035.411} C_VEL
LIN {X 0,Y 539.299,Z 530.815,A -85,B 0,C 180,E1 -4036.745,E2 -4036.745} C_VEL
LIN {X 0,Y 539.135,Z 544.103,A -85,B 0,C 180,E1 -4037.077,E2 -4037.077} C_VEL
LIN {X 0,Y 538.944,Z 556.275,A -85,B 0,C 180,E1 -4037.527,E2 -4037.527} C_VEL
LIN {X 0,Y 538.692,Z 568.119,A -85,B 0,C 180,E1 -4038.116,E2 -4038.116} C_VEL
LIN {X 0,Y 538.526,Z 580.155,A -85,B 0,C 180,E1 -4038.901,E2 -4038.901} C_VEL
LIN {X 0,Y 538.263,Z 590.597,A -85,B 0,C 180,E1 -4039.752,E2 -4039.752} C_VEL
LIN {X 0,Y 538.067,Z 599.111,A -85,B 0,C 180,E1 -4040.603,E2 -4040.603} C_VEL
LIN {X 0,Y 537.921,Z 606.959,A -85,B 0,C 180,E1 -4041.548,E2 -4041.548} C_VEL
LIN {X 0,Y 537.755,Z 614.62,A -85,B 0,C 180,E1 -4042.679,E2 -4042.679} C_VEL
LIN {X 0,Y 537.693,Z 621.678,A -85,B 0,C 180,E1 -4043.998,E2 -4043.998} C_VEL
LIN {X 0,Y 537.541,Z 626.372,A -85,B 0,C 180,E1 -4045.125,E2 -4045.125} C_VEL
LIN {X 0,Y 537.591,Z 629.957,A -85,B 0,C 180,E1 -4046.252,E2 -4046.252} C_VEL
LIN {X 0,Y 537.551,Z 631.806,A -85,B 0,C 180,E1 -4047.002,E2 -4047.002} C_VEL
LIN {X 0,Y 537.451,Z 634.182,A -85,B 0,C 180,E1 -4048.501,E2 -4048.501} C_VEL
LIN {X 0,Y 537.442,Z 635,A -85,B 0,C 180,E1 -4050,E2 -4050} C_VEL
LIN {X 0,Y 537.451,Z 634.184,A -85,B 0,C 180,E1 -4051.498,E2 -4051.498} C_VEL
LIN {X 0,Y 537.551,Z 631.81,A -85,B 0,C 180,E1 -4052.998,E2 -4052.998} C_VEL
LIN {X 0,Y 537.603,Z 628.895,A -85,B 0,C 180,E1 -4054.123,E2 -4054.123} C_VEL
LIN {X 0,Y 537.588,Z 624.948,A -85,B 0,C 180,E1 -4055.251,E2 -4055.251} C_VEL
LIN {X 0,Y 537.644,Z 620.125,A -85,B 0,C 180,E1 -4056.326,E2 -4056.326} C_VEL
LIN {X 0,Y 537.791,Z 613.467,A -85,B 0,C 180,E1 -4057.509,E2 -4057.509} C_VEL
LIN {X 0,Y 537.972,Z 605.478,A -85,B 0,C 180,E1 -4058.64,E2 -4058.64} C_VEL
LIN {X 0,Y 538.143,Z 597.333,A -85,B 0,C 180,E1 -4059.585,E2 -4059.585} C_VEL
LIN {X 0,Y 538.384,Z 587.384,A -85,B 0,C 180,E1 -4060.53,E2 -4060.53} C_VEL
LIN {X 0,Y 538.565,Z 577.551,A -85,B 0,C 180,E1 -4061.288,E2 -4061.288} C_VEL
LIN {X 0,Y 538.754,Z 566.476,A -85,B 0,C 180,E1 -4061.973,E2 -4061.973} C_VEL
LIN {X 0,Y 538.962,Z 554.01,A -85,B 0,C 180,E1 -4062.568,E2 -4062.568} C_VEL
LIN {X 0,Y 539.21,Z 540.979,A -85,B 0,C 180,E1 -4063.017,E2 -4063.017} C_VEL
LIN {X 0,Y 539.324,Z 527.984,A -85,B 0,C 180,E1 -4063.302,E2 -4063.302} C_VEL
LIN {X 0,Y 539.554,Z 430.65,A -85,B 0,C 180,E1 -4064.611,E2 -4064.611} C_VEL
LIN {X 0,Y 538.327,Z 422.838,A -85,B 0,C 180,E1 -4064.75,E2 -4064.75} C_VEL
LIN {X 0,Y 538.709,Z 401.329,A -85,B 0,C 180,E1 -4068.087,E2 -4068.087} C_VEL
LIN {X 0,Y 539.094,Z 381.557,A -85,B 0,C 180,E1 -4071.209,E2 -4071.209} C_VEL
LIN {X 0,Y 539.162,Z 372.792,A -85,B 0,C 180,E1 -4072.614,E2 -4072.614} C_VEL
LIN {X 0,Y 538.056,Z 366.965,A -85,B 0,C 180,E1 -4073.628,E2 -4073.628} C_VEL
LIN {X 0,Y 538.045,Z 366.96,A -85,B 0,C 180,E1 -4076.366,E2 -4076.366} C_VEL
LIN {X 0,Y 538.034,Z 366.968,A -85,B 0,C 180,E1 -4078.934,E2 -4078.934} C_VEL
LIN {X 0,Y 538.031,Z 366.961,A -85,B 0,C 180,E1 -4081.89,E2 -4081.89} C_VEL
LIN {X 0,Y 538.028,Z 366.963,A -85,B 0,C 180,E1 -4084.62,E2 -4084.62} C_VEL
LIN {X 0,Y 538.007,Z 366.97,A -85,B 0,C 180,E1 -4087.17,E2 -4087.17} C_VEL
LIN {X 0,Y 538.03,Z 366.961,A -85,B 0,C 180,E1 -4089.796,E2 -4089.796} C_VEL
LIN {X 0,Y 538.021,Z 366.968,A -85,B 0,C 180,E1 -4092.786,E2 -4092.786} C_VEL
LIN {X 0,Y 538.035,Z 366.965,A -85,B 0,C 180,E1 -4095.141,E2 -4095.141} C_VEL
LIN {X 0,Y 538.042,Z 366.96,A -85,B 0,C 180,E1 -4098.228,E2 -4098.228} C_VEL
LIN {X 0,Y 538.015,Z 366.966,A -85,B 0,C 180,E1 -4101.17,E2 -4101.17} C_VEL
LIN {X 0,Y 537.996,Z 366.965,A -85,B 0,C 180,E1 -4104.089,E2 -4104.089} C_VEL
LIN {X 0,Y 538.033,Z 366.97,A -85,B 0,C 180,E1 -4106.727,E2 -4106.727} C_VEL
LIN {X 0,Y 538.029,Z 366.96,A -85,B 0,C 180,E1 -4109.556,E2 -4109.556} C_VEL
LIN {X 0,Y 538.047,Z 366.959,A -85,B 0,C 180,E1 -4111.95,E2 -4111.95} C_VEL
LIN {X 0,Y 538.074,Z 366.962,A -85,B 0,C 180,E1 -4114.467,E2 -4114.467} C_VEL
LIN {X 0,Y 537.997,Z 366.965,A -85,B 0,C 180,E1 -4117.738,E2 -4117.738} C_VEL
LIN {X 0,Y 538.083,Z 366.957,A -85,B 0,C 180,E1 -4120.148,E2 -4120.148} C_VEL
LIN {X 0,Y 538.027,Z 366.961,A -85,B 0,C 180,E1 -4123.299,E2 -4123.299} C_VEL
LIN {X 0,Y 538.067,Z 366.956,A -85,B 0,C 180,E1 -4125.631,E2 -4125.631} C_VEL
LIN {X 0,Y 538.081,Z 366.959,A -85,B 0,C 180,E1 -4128.702,E2 -4128.702} C_VEL
LIN {X 0,Y 538.066,Z 366.957,A -85,B 0,C 180,E1 -4131.739,E2 -4131.739} C_VEL
LIN {X 0,Y 538.125,Z 366.953,A -85,B 0,C 180,E1 -4134.003,E2 -4134.003} C_VEL
LIN {X 0,Y 538.142,Z 366.947,A -85,B 0,C 180,E1 -4137.006,E2 -4137.006} C_VEL
LIN {X 0,Y 538.177,Z 366.948,A -85,B 0,C 180,E1 -4140,E2 -4140} C_VEL
LIN {X 0,Y 538.143,Z 366.946,A -85,B 0,C 180,E1 -4142.994,E2 -4142.994} C_VEL
LIN {X 0,Y 538.127,Z 366.956,A -85,B 0,C 180,E1 -4145.997,E2 -4145.997} C_VEL
LIN {X 0,Y 538.065,Z 366.956,A -85,B 0,C 180,E1 -4149.018,E2 -4149.018} C_VEL
LIN {X 0,Y 538.087,Z 366.962,A -85,B 0,C 180,E1 -4152.063,E2 -4152.063} C_VEL
LIN {X 0,Y 538.05,Z 366.958,A -85,B 0,C 180,E1 -4155.144,E2 -4155.144} C_VEL
LIN {X 0,Y 538.038,Z 366.964,A -85,B 0,C 180,E1 -4158.27,E2 -4158.27} C_VEL
LIN {X 0,Y 538.043,Z 366.959,A -85,B 0,C 180,E1 -4160.651,E2 -4160.651} C_VEL
LIN {X 0,Y 538.028,Z 366.969,A -85,B 0,C 180,E1 -4163.887,E2 -4163.887} C_VEL
LIN {X 0,Y 538.046,Z 366.96,A -85,B 0,C 180,E1 -4166.367,E2 -4166.367} C_VEL
LIN {X 0,Y 538.034,Z 366.96,A -85,B 0,C 180,E1 -4168.934,E2 -4168.934} C_VEL
LIN {X 0,Y 538.018,Z 366.968,A -85,B 0,C 180,E1 -4171.888,E2 -4171.888} C_VEL
LIN {X 0,Y 538.03,Z 366.96,A -85,B 0,C 180,E1 -4174.62,E2 -4174.62} C_VEL
LIN {X 0,Y 538.011,Z 366.965,A -85,B 0,C 180,E1 -4177.171,E2 -4177.171} C_VEL
LIN {X 0,Y 538.021,Z 366.962,A -85,B 0,C 180,E1 -4180.262,E2 -4180.262} C_VEL
LIN {X 0,Y 537.373,Z 367.043,A -85,B 0,C 180,E1 -4180.887,E2 -4180.887} C_VEL
LIN {X 0,Y 534.526,Z 367.406,A -85,B 0,C 180,E1 -4181.902,E2 -4181.902} C_VEL
LIN {X 0,Y 532.104,Z 367.713,A -85,B 0,C 180,E1 -4182.719,E2 -4182.719} C_VEL
LIN {X 0,Y 531.056,Z 367.84,A -85,B 0,C 180,E1 -4183.351,E2 -4183.351} C_VEL
LIN {X 0,Y 530.968,Z 367.848,A -85,B 0,C 180,E1 -4183.564,E2 -4183.564} C_VEL
LIN {X 0,Y 530.968,Z 367.84,A -85,B 0,C 180,E1 -4186.506,E2 -4186.506} C_VEL
LIN {X 0,Y 530.987,Z 367.845,A -85,B 0,C 180,E1 -4189.567,E2 -4189.567} C_VEL
LIN {X 0,Y 530.972,Z 367.84,A -85,B 0,C 180,E1 -4192.577,E2 -4192.577} C_VEL
LIN {X 0,Y 531.005,Z 367.844,A -85,B 0,C 180,E1 -4195.311,E2 -4195.311} C_VEL
LIN {X 0,Y 530.97,Z 367.84,A -85,B 0,C 180,E1 -4198.032,E2 -4198.032} C_VEL
LIN {X 0,Y 530.992,Z 367.841,A -85,B 0,C 180,E1 -4200.874,E2 -4200.874} C_VEL
LIN {X 0,Y 531.005,Z 367.845,A -85,B 0,C 180,E1 -4203.256,E2 -4203.256} C_VEL
LIN {X 0,Y 530.987,Z 367.841,A -85,B 0,C 180,E1 -4205.961,E2 -4205.961} C_VEL
LIN {X 0,Y 531.04,Z 367.938,A -85,B 0,C 180,E1 -4209.165,E2 -4209.165} C_VEL
LIN {X 0,Y 531.723,Z 372.688,A -85,B 0,C 180,E1 -4210.102,E2 -4210.102} C_VEL
LIN {X 0,Y 531.507,Z 386.46,A -85,B 0,C 180,E1 -4212.692,E2 -4212.692} C_VEL
LIN {X 0,Y 531.248,Z 399.426,A -85,B 0,C 180,E1 -4215.1,E2 -4215.1} C_VEL
LIN {X 0,Y 532.842,Z 409.999,A -85,B 0,C 180,E1 -4215.298,E2 -4215.298} C_VEL
LIN {X 0,Y 532.476,Z 506.444,A -85,B 0,C 180,E1 -4216.621,E2 -4216.621} C_VEL
LIN {X 0,Y 532.263,Z 519.637,A -85,B 0,C 180,E1 -4216.956,E2 -4216.956} C_VEL
LIN {X 0,Y 532.047,Z 531.743,A -85,B 0,C 180,E1 -4217.411,E2 -4217.411} C_VEL
LIN {X 0,Y 531.841,Z 543.628,A -85,B 0,C 180,E1 -4218.016,E2 -4218.016} C_VEL
LIN {X 0,Y 531.561,Z 554.845,A -85,B 0,C 180,E1 -4218.754,E2 -4218.754} C_VEL
LIN {X 0,Y 531.29,Z 565.329,A -85,B 0,C 180,E1 -4219.617,E2 -4219.617} C_VEL
LIN {X 0,Y 531.071,Z 573.894,A -85,B 0,C 180,E1 -4220.478,E2 -4220.478} C_VEL
LIN {X 0,Y 530.891,Z 581.783,A -85,B 0,C 180,E1 -4221.435,E2 -4221.435} C_VEL
LIN {X 0,Y 530.723,Z 589.498,A -85,B 0,C 180,E1 -4222.582,E2 -4222.582} C_VEL
LIN {X 0,Y 530.606,Z 596.573,A -85,B 0,C 180,E1 -4223.918,E2 -4223.918} C_VEL
LIN {X 0,Y 530.459,Z 601.291,A -85,B 0,C 180,E1 -4225.06,E2 -4225.06} C_VEL
LIN {X 0,Y 530.516,Z 604.901,A -85,B 0,C 180,E1 -4226.202,E2 -4226.202} C_VEL
LIN {X 0,Y 530.457,Z 606.769,A -85,B 0,C 180,E1 -4226.962,E2 -4226.962} C_VEL
LIN {X 0,Y 530.411,Z 608.18,A -85,B 0,C 180,E1 -4227.722,E2 -4227.722} C_VEL
LIN {X 0,Y 530.344,Z 609.801,A -85,B 0,C 180,E1 -4229.241,E2 -4229.241} C_VEL
LIN {X 0,Y 530.343,Z 610.039,A -85,B 0,C 180,E1 -4230,E2 -4230} C_VEL
LIN {X 0,Y 530.344,Z 609.857,A -85,B 0,C 180,E1 -4230.759,E2 -4230.759} C_VEL
LIN {X 0,Y 530.411,Z 608.309,A -85,B 0,C 180,E1 -4232.278,E2 -4232.278} C_VEL
LIN {X 0,Y 530.457,Z 606.954,A -85,B 0,C 180,E1 -4233.038,E2 -4233.038} C_VEL
LIN {X 0,Y 530.523,Z 604.09,A -85,B 0,C 180,E1 -4234.178,E2 -4234.178} C_VEL
LIN {X 0,Y 530.524,Z 600.208,A -85,B 0,C 180,E1 -4235.321,E2 -4235.321} C_VEL
LIN {X 0,Y 530.593,Z 594.649,A -85,B 0,C 180,E1 -4236.576,E2 -4236.576} C_VEL
LIN {X 0,Y 530.779,Z 587.668,A -85,B 0,C 180,E1 -4237.8,E2 -4237.8} C_VEL
LIN {X 0,Y 530.907,Z 579.517,A -85,B 0,C 180,E1 -4238.949,E2 -4238.949} C_VEL
LIN {X 0,Y 531.12,Z 571.173,A -85,B 0,C 180,E1 -4239.906,E2 -4239.906} C_VEL
LIN {X 0,Y 531.396,Z 560.873,A -85,B 0,C 180,E1 -4240.863,E2 -4240.863} C_VEL
LIN {X 0,Y 531.671,Z 549.062,A -85,B 0,C 180,E1 -4241.739,E2 -4241.739} C_VEL
LIN {X 0,Y 531.942,Z 537.697,A -85,B 0,C 180,E1 -4242.398,E2 -4242.398} C_VEL
LIN {X 0,Y 532.175,Z 525.683,A -85,B 0,C 180,E1 -4242.925,E2 -4242.925} C_VEL
LIN {X 0,Y 532.355,Z 512.617,A -85,B 0,C 180,E1 -4243.334,E2 -4243.334} C_VEL
LIN {X 0,Y 532.498,Z 500.148,A -85,B 0,C 180,E1 -4243.573,E2 -4243.573} C_VEL
LIN {X 0,Y 532.721,Z 408.203,A -85,B 0,C 180,E1 -4244.82,E2 -4244.82} C_VEL
LIN {X 0,Y 531.241,Z 399.424,A -85,B 0,C 180,E1 -4244.993,E2 -4244.993} C_VEL
LIN {X 0,Y 531.597,Z 382.914,A -85,B 0,C 180,E1 -4248.061,E2 -4248.061} C_VEL
LIN {X 0,Y 531.668,Z 371.626,A -85,B 0,C 180,E1 -4250.193,E2 -4250.193} C_VEL
LIN {X 0,Y 531.021,Z 367.843,A -85,B 0,C 180,E1 -4250.988,E2 -4250.988} C_VEL
LIN {X 0,Y 530.975,Z 367.844,A -85,B 0,C 180,E1 -4254.225,E2 -4254.225} C_VEL
LIN {X 0,Y 531.005,Z 367.844,A -85,B 0,C 180,E1 -4256.744,E2 -4256.744} C_VEL
LIN {X 0,Y 530.986,Z 367.84,A -85,B 0,C 180,E1 -4259.323,E2 -4259.323} C_VEL
LIN {X 0,Y 530.97,Z 367.841,A -85,B 0,C 180,E1 -4262.1,E2 -4262.1} C_VEL
LIN {X 0,Y 530.983,Z 367.846,A -85,B 0,C 180,E1 -4264.852,E2 -4264.852} C_VEL
LIN {X 0,Y 530.97,Z 367.84,A -85,B 0,C 180,E1 -4267.508,E2 -4267.508} C_VEL
LIN {X 0,Y 530.985,Z 367.844,A -85,B 0,C 180,E1 -4270.433,E2 -4270.433} C_VEL
LIN {X 0,Y 530.965,Z 367.841,A -85,B 0,C 180,E1 -4273.281,E2 -4273.281} C_VEL
LIN {X 0,Y 530.993,Z 367.837,A -85,B 0,C 180,E1 -4275.621,E2 -4275.621} C_VEL
LIN {X 0,Y 531.003,Z 367.844,A -85,B 0,C 180,E1 -4278.565,E2 -4278.565} C_VEL
LIN {X 0,Y 530.96,Z 367.841,A -85,B 0,C 180,E1 -4281.529,E2 -4281.529} C_VEL
LIN {X 0,Y 530.959,Z 367.85,A -85,B 0,C 180,E1 -4284.38,E2 -4284.38} C_VEL
LIN {X 0,Y 530.972,Z 367.84,A -85,B 0,C 180,E1 -4287.134,E2 -4287.134} C_VEL
LIN {X 0,Y 530.975,Z 367.841,A -85,B 0,C 180,E1 -4289.803,E2 -4289.803} C_VEL
LIN {X 0,Y 531.021,Z 367.84,A -85,B 0,C 180,E1 -4292.467,E2 -4292.467} C_VEL
LIN {X 0,Y 531.001,Z 367.837,A -85,B 0,C 180,E1 -4294.942,E2 -4294.942} C_VEL
LIN {X 0,Y 530.977,Z 367.847,A -85,B 0,C 180,E1 -4298.247,E2 -4298.247} C_VEL
LIN {X 0,Y 531,Z 367.838,A -85,B 0,C 180,E1 -4300.677,E2 -4300.677} C_VEL
LIN {X 0,Y 530.991,Z 367.837,A -85,B 0,C 180,E1 -4303.071,E2 -4303.071} C_VEL
LIN {X 0,Y 531.026,Z 367.834,A -85,B 0,C 180,E1 -4305.436,E2 -4305.436} C_VEL
LIN {X 0,Y 531.043,Z 367.833,A -85,B 0,C 180,E1 -4308.55,E2 -4308.55} C_VEL
LIN {X 0,Y 531.059,Z 367.833,A -85,B 0,C 180,E1 -4311.629,E2 -4311.629} C_VEL
LIN {X 0,Y 531.126,Z 367.821,A -85,B 0,C 180,E1 -4314.685,E2 -4314.685} C_VEL
LIN {X 0,Y 531.145,Z 367.825,A -85,B 0,C 180,E1 -4317.725,E2 -4317.725} C_VEL
LIN {X 0,Y 531.158,Z 367.816,A -85,B 0,C 180,E1 -4320.758,E2 -4320.758} C_VEL
LIN {X 0,Y 531.111,Z 367.823,A -85,B 0,C 180,E1 -4323.034,E2 -4323.034} C_VEL
LIN {X 0,Y 531.09,Z 367.829,A -85,B 0,C 180,E1 -4326.077,E2 -4326.077} C_VEL
LIN {X 0,Y 531.021,Z 367.835,A -85,B 0,C 180,E1 -4329.138,E2 -4329.138} C_VEL
LIN {X 0,Y 531.046,Z 367.832,A -85,B 0,C 180,E1 -4332.225,E2 -4332.225} C_VEL
LIN {X 0,Y 531.001,Z 367.842,A -85,B 0,C 180,E1 -4335.35,E2 -4335.35} C_VEL
LIN {X 0,Y 530.992,Z 367.837,A -85,B 0,C 180,E1 -4338.521,E2 -4338.521} C_VEL
LIN {X 0,Y 531.005,Z 367.837,A -85,B 0,C 180,E1 -4340.938,E2 -4340.938} C_VEL
LIN {X 0,Y 530.971,Z 367.84,A -85,B 0,C 180,E1 -4344.225,E2 -4344.225} C_VEL
LIN {X 0,Y 531.003,Z 367.837,A -85,B 0,C 180,E1 -4346.744,E2 -4346.744} C_VEL
LIN {X 0,Y 530.986,Z 367.847,A -85,B 0,C 180,E1 -4349.322,E2 -4349.322} C_VEL
LIN {X 0,Y 530.97,Z 367.84,A -85,B 0,C 180,E1 -4352.1,E2 -4352.1} C_VEL
LIN {X 0,Y 530.972,Z 367.843,A -85,B 0,C 180,E1 -4354.85,E2 -4354.85} C_VEL
LIN {X 0,Y 530.969,Z 367.845,A -85,B 0,C 180,E1 -4357.508,E2 -4357.508} C_VEL
LIN {X 0,Y 530.985,Z 367.839,A -85,B 0,C 180,E1 -4360.433,E2 -4360.433} C_VEL
LIN {X 0,Y 530.969,Z 367.844,A -85,B 0,C 180,E1 -4363.494,E2 -4363.494} C_VEL
LIN {X 0,Y 530.958,Z 367.843,A -85,B 0,C 180,E1 -4366.504,E2 -4366.504} C_VEL
LIN {X 0,Y 530.988,Z 367.846,A -85,B 0,C 180,E1 -4368.976,E2 -4368.976} C_VEL
LIN {X 0,Y 530.963,Z 367.843,A -85,B 0,C 180,E1 -4371.529,E2 -4371.529} C_VEL
LIN {X 0,Y 530.962,Z 367.842,A -85,B 0,C 180,E1 -4374.38,E2 -4374.38} C_VEL
LIN {X 0,Y 530.971,Z 367.845,A -85,B 0,C 180,E1 -4377.133,E2 -4377.133} C_VEL
LIN {X 0,Y 530.974,Z 367.841,A -85,B 0,C 180,E1 -4379.803,E2 -4379.803} C_VEL
LIN {X 0,Y 531.017,Z 367.84,A -85,B 0,C 180,E1 -4382.467,E2 -4382.467} C_VEL
LIN {X 0,Y 531.01,Z 367.844,A -85,B 0,C 180,E1 -4384.942,E2 -4384.942} C_VEL
LIN {X 0,Y 530.992,Z 367.875,A -85,B 0,C 180,E1 -4386.236,E2 -4386.236} C_VEL
LIN {X 0,Y 532.308,Z 375.533,A -85,B 0,C 180,E1 -4387.549,E2 -4387.549} C_VEL
LIN {X 0,Y 531.922,Z 391.42,A -85,B 0,C 180,E1 -4390.109,E2 -4390.109} C_VEL
LIN {X 0,Y 531.559,Z 408.937,A -85,B 0,C 180,E1 -4392.891,E2 -4392.891} C_VEL
LIN {X 0,Y 531.303,Z 422.673,A -85,B 0,C 180,E1 -4395.048,E2 -4395.048} C_VEL
LIN {X 0,Y 532.819,Z 432.54,A -85,B 0,C 180,E1 -4395.229,E2 -4395.229} C_VEL
LIN {X 0,Y 532.397,Z 530.648,A -85,B 0,C 180,E1 -4396.57,E2 -4396.57} C_VEL
LIN {X 0,Y 532.206,Z 543.935,A -85,B 0,C 180,E1 -4396.905,E2 -4396.905} C_VEL
LIN {X 0,Y 531.985,Z 556.107,A -85,B 0,C 180,E1 -4397.361,E2 -4397.361} C_VEL
LIN {X 0,Y 531.714,Z 568.461,A -85,B 0,C 180,E1 -4397.989,E2 -4397.989} C_VEL
LIN {X 0,Y 531.507,Z 579.986,A -85,B 0,C 180,E1 -4398.753,E2 -4398.753} C_VEL
LIN {X 0,Y 531.224,Z 590.428,A -85,B 0,C 180,E1 -4399.615,E2 -4399.615} C_VEL
LIN {X 0,Y 531.033,Z 598.966,A -85,B 0,C 180,E1 -4400.477,E2 -4400.477} C_VEL
LIN {X 0,Y 530.887,Z 606.844,A -85,B 0,C 180,E1 -4401.435,E2 -4401.435} C_VEL
LIN {X 0,Y 530.682,Z 614.535,A -85,B 0,C 180,E1 -4402.581,E2 -4402.581} C_VEL
LIN {X 0,Y 530.604,Z 621.627,A -85,B 0,C 180,E1 -4403.917,E2 -4403.917} C_VEL
LIN {X 0,Y 530.459,Z 626.341,A -85,B 0,C 180,E1 -4405.06,E2 -4405.06} C_VEL
LIN {X 0,Y 530.516,Z 629.947,A -85,B 0,C 180,E1 -4406.202,E2 -4406.202} C_VEL
LIN {X 0,Y 530.457,Z 631.803,A -85,B 0,C 180,E1 -4406.962,E2 -4406.962} C_VEL
LIN {X 0,Y 530.41,Z 633.192,A -85,B 0,C 180,E1 -4407.722,E2 -4407.722} C_VEL
LIN {X 0,Y 530.344,Z 634.785,A -85,B 0,C 180,E1 -4409.241,E2 -4409.241} C_VEL
LIN {X 0,Y 530.342,Z 635,A -85,B 0,C 180,E1 -4410,E2 -4410} C_VEL
LIN {X 0,Y 530.361,Z 634.183,A -85,B 0,C 180,E1 -4411.519,E2 -4411.519} C_VEL
LIN {X 0,Y 530.41,Z 633.195,A -85,B 0,C 180,E1 -4412.278,E2 -4412.278} C_VEL
LIN {X 0,Y 530.457,Z 631.807,A -85,B 0,C 180,E1 -4413.038,E2 -4413.038} C_VEL
LIN {X 0,Y 530.522,Z 628.879,A -85,B 0,C 180,E1 -4414.178,E2 -4414.178} C_VEL
LIN {X 0,Y 530.525,Z 624.911,A -85,B 0,C 180,E1 -4415.321,E2 -4415.321} C_VEL
LIN {X 0,Y 530.596,Z 619.215,A -85,B 0,C 180,E1 -4416.579,E2 -4416.579} C_VEL
LIN {X 0,Y 530.737,Z 612.141,A -85,B 0,C 180,E1 -4417.801,E2 -4417.801} C_VEL
LIN {X 0,Y 530.93,Z 603.866,A -85,B 0,C 180,E1 -4418.948,E2 -4418.948} C_VEL
LIN {X 0,Y 531.131,Z 595.384,A -85,B 0,C 180,E1 -4419.905,E2 -4419.905} C_VEL
LIN {X 0,Y 531.397,Z 584.902,A -85,B 0,C 180,E1 -4420.863,E2 -4420.863} C_VEL
LIN {X 0,Y 531.664,Z 572.946,A -85,B 0,C 180,E1 -4421.737,E2 -4421.737} C_VEL
LIN {X 0,Y 531.936,Z 561.241,A -85,B 0,C 180,E1 -4422.398,E2 -4422.398} C_VEL
LIN {X 0,Y 532.125,Z 548.898,A -85,B 0,C 180,E1 -4422.926,E2 -4422.926} C_VEL
LIN {X 0,Y 532.346,Z 536.235,A -85,B 0,C 180,E1 -4423.309,E2 -4423.309} C_VEL
LIN {X 0,Y 532.493,Z 523.022,A -85,B 0,C 180,E1 -4423.549,E2 -4423.549} C_VEL
LIN {X 0,Y 532.673,Z 431.347,A -85,B 0,C 180,E1 -4424.792,E2 -4424.792} C_VEL
LIN {X 0,Y 531.325,Z 422.612,A -85,B 0,C 180,E1 -4424.961,E2 -4424.961} C_VEL
LIN {X 0,Y 531.716,Z 401.346,A -85,B 0,C 180,E1 -4428.307,E2 -4428.307} C_VEL
LIN {X 0,Y 532.146,Z 382.665,A -85,B 0,C 180,E1 -4431.296,E2 -4431.296} C_VEL
LIN {X 0,Y 532.29,Z 375.152,A -85,B 0,C 180,E1 -4432.513,E2 -4432.513} C_VEL
LIN {X 0,Y 530.99,Z 367.844,A -85,B 0,C 180,E1 -4433.812,E2 -4433.812} C_VEL
LIN {X 0,Y 531.008,Z 367.84,A -85,B 0,C 180,E1 -4436.744,E2 -4436.744} C_VEL
LIN {X 0,Y 530.985,Z 367.845,A -85,B 0,C 180,E1 -4439.322,E2 -4439.322} C_VEL
LIN {X 0,Y 530.983,Z 367.838,A -85,B 0,C 180,E1 -4442.103,E2 -4442.103} C_VEL
LIN {X 0,Y 530.983,Z 367.844,A -85,B 0,C 180,E1 -4444.853,E2 -4444.853} C_VEL
LIN {X 0,Y 530.968,Z 367.843,A -85,B 0,C 180,E1 -4447.508,E2 -4447.508} C_VEL
LIN {X 0,Y 530.986,Z 367.84,A -85,B 0,C 180,E1 -4450.433,E2 -4450.433} C_VEL
LIN {X 0,Y 530.967,Z 367.842,A -85,B 0,C 180,E1 -4453.494,E2 -4453.494} C_VEL
LIN {X 0,Y 530.969,Z 367.843,A -85,B 0,C 180,E1 -4456.506,E2 -4456.506} C_VEL
LIN {X 0,Y 530.99,Z 367.845,A -85,B 0,C 180,E1 -4458.976,E2 -4458.976} C_VEL
LIN {X 0,Y 530.959,Z 367.842,A -85,B 0,C 180,E1 -4461.529,E2 -4461.529} C_VEL
LIN {X 0,Y 530.956,Z 367.845,A -85,B 0,C 180,E1 -4464.38,E2 -4464.38} C_VEL
LIN {X 0,Y 530.97,Z 367.843,A -85,B 0,C 180,E1 -4467.133,E2 -4467.133} C_VEL
LIN {X 0,Y 530.972,Z 367.84,A -85,B 0,C 180,E1 -4469.803,E2 -4469.803} C_VEL
LIN {X 0,Y 531.018,Z 367.84,A -85,B 0,C 180,E1 -4472.467,E2 -4472.467} C_VEL
LIN {X 0,Y 530.998,Z 367.84,A -85,B 0,C 180,E1 -4474.942,E2 -4474.942} C_VEL
LIN {X 0,Y 530.975,Z 367.844,A -85,B 0,C 180,E1 -4478.247,E2 -4478.247} C_VEL
LIN {X 0,Y 530.998,Z 367.843,A -85,B 0,C 180,E1 -4480.677,E2 -4480.677} C_VEL
LIN {X 0,Y 530.989,Z 367.839,A -85,B 0,C 180,E1 -4483.071,E2 -4483.071} C_VEL
LIN {X 0,Y 531.023,Z 367.833,A -85,B 0,C 180,E1 -4485.436,E2 -4485.436} C_VEL
LIN {X 0,Y 531.053,Z 367.836,A -85,B 0,C 180,E1 -4488.55,E2 -4488.55} C_VEL
LIN {X 0,Y 531.041,Z 367.832,A -85,B 0,C 180,E1 -4491.629,E2 -4491.629} C_VEL
LIN {X 0,Y 531.123,Z 367.824,A -85,B 0,C 180,E1 -4494.685,E2 -4494.685} C_VEL
LIN {X 0,Y 531.142,Z 367.821,A -85,B 0,C 180,E1 -4497.725,E2 -4497.725} C_VEL
LIN {X 0,Y 531.156,Z 367.818,A -85,B 0,C 180,E1 -4500.758,E2 -4500.758} C_VEL
LIN {X 0,Y 531.109,Z 367.822,A -85,B 0,C 180,E1 -4503.034,E2 -4503.034} C_VEL
LIN {X 0,Y 531.087,Z 367.834,A -85,B 0,C 180,E1 -4506.077,E2 -4506.077} C_VEL
LIN {X 0,Y 531.057,Z 367.834,A -85,B 0,C 180,E1 -4508.371,E2 -4508.371} C_VEL
LIN {X 0,Y 531.055,Z 367.833,A -85,B 0,C 180,E1 -4511.672,E2 -4511.672} C_VEL
LIN {X 0,Y 531.035,Z 367.832,A -85,B 0,C 180,E1 -4514.956,E2 -4514.956} C_VEL
LIN {X 0,Y 531.021,Z 367.839,A -85,B 0,C 180,E1 -4517.722,E2 -4517.722} C_VEL
LIN {X 0,Y 531.004,Z 367.836,A -85,B 0,C 180,E1 -4520.938,E2 -4520.938} C_VEL
LIN {X 0,Y 530.984,Z 367.842,A -85,B 0,C 180,E1 -4524.224,E2 -4524.224} C_VEL
LIN {X 0,Y 531.009,Z 367.835,A -85,B 0,C 180,E1 -4526.744,E2 -4526.744} C_VEL
LIN {X 0,Y 530.985,Z 367.841,A -85,B 0,C 180,E1 -4529.323,E2 -4529.323} C_VEL
LIN {X 0,Y 530.974,Z 367.843,A -85,B 0,C 180,E1 -4532.101,E2 -4532.101} C_VEL
LIN {X 0,Y 530.988,Z 367.838,A -85,B 0,C 180,E1 -4534.853,E2 -4534.853} C_VEL
LIN {X 0,Y 530.97,Z 367.847,A -85,B 0,C 180,E1 -4537.508,E2 -4537.508} C_VEL
LIN {X 0,Y 530.985,Z 367.838,A -85,B 0,C 180,E1 -4540.433,E2 -4540.433} C_VEL
LIN {X 0,Y 530.971,Z 367.849,A -85,B 0,C 180,E1 -4543.494,E2 -4543.494} C_VEL
LIN {X 0,Y 530.968,Z 367.848,A -85,B 0,C 180,E1 -4543.564,E2 -4543.564} C_VEL
LIN {X 0,Y 530.294,Z 367.926,A -85,B 0,C 180,E1 -4544.198,E2 -4544.198} C_VEL
LIN {X 0,Y 527.445,Z 368.284,A -85,B 0,C 180,E1 -4545.227,E2 -4545.227} C_VEL
LIN {X 0,Y 525.041,Z 368.581,A -85,B 0,C 180,E1 -4546.055,E2 -4546.055} C_VEL
LIN {X 0,Y 524.007,Z 368.708,A -85,B 0,C 180,E1 -4546.695,E2 -4546.695} C_VEL
LIN {X 0,Y 523.922,Z 368.719,A -85,B 0,C 180,E1 -4546.911,E2 -4546.911} C_VEL
LIN {X 0,Y 523.951,Z 368.717,A -85,B 0,C 180,E1 -4549.921,E2 -4549.921} C_VEL
LIN {X 0,Y 523.915,Z 368.721,A -85,B 0,C 180,E1 -4552.868,E2 -4552.868} C_VEL
LIN {X 0,Y 523.948,Z 368.718,A -85,B 0,C 180,E1 -4555.711,E2 -4555.711} C_VEL
LIN {X 0,Y 523.924,Z 368.718,A -85,B 0,C 180,E1 -4558.456,E2 -4558.456} C_VEL
LIN {X 0,Y 523.942,Z 368.722,A -85,B 0,C 180,E1 -4561.125,E2 -4561.125} C_VEL
LIN {X 0,Y 523.987,Z 368.712,A -85,B 0,C 180,E1 -4563.98,E2 -4563.98} C_VEL
LIN {X 0,Y 523.928,Z 368.72,A -85,B 0,C 180,E1 -4566.27,E2 -4566.27} C_VEL
LIN {X 0,Y 524.011,Z 368.871,A -85,B 0,C 180,E1 -4569.027,E2 -4569.027} C_VEL
LIN {X 0,Y 524.777,Z 374.06,A -85,B 0,C 180,E1 -4570.065,E2 -4570.065} C_VEL
LIN {X 0,Y 524.52,Z 387.662,A -85,B 0,C 180,E1 -4572.655,E2 -4572.655} C_VEL
LIN {X 0,Y 524.248,Z 399.621,A -85,B 0,C 180,E1 -4574.9,E2 -4574.9} C_VEL
LIN {X 0,Y 525.983,Z 410,A -85,B 0,C 180,E1 -4575.099,E2 -4575.099} C_VEL
LIN {X 0,Y 525.597,Z 506.64,A -85,B 0,C 180,E1 -4576.443,E2 -4576.443} C_VEL
LIN {X 0,Y 525.347,Z 519.824,A -85,B 0,C 180,E1 -4576.781,E2 -4576.781} C_VEL
LIN {X 0,Y 525.111,Z 531.925,A -85,B 0,C 180,E1 -4577.242,E2 -4577.242} C_VEL
LIN {X 0,Y 524.932,Z 542.572,A -85,B 0,C 180,E1 -4577.784,E2 -4577.784} C_VEL
LIN {X 0,Y 524.618,Z 553.734,A -85,B 0,C 180,E1 -4578.506,E2 -4578.506} C_VEL
LIN {X 0,Y 524.341,Z 564.437,A -85,B 0,C 180,E1 -4579.38,E2 -4579.38} C_VEL
LIN {X 0,Y 524.069,Z 574.067,A -85,B 0,C 180,E1 -4580.35,E2 -4580.35} C_VEL
LIN {X 0,Y 523.868,Z 581.955,A -85,B 0,C 180,E1 -4581.32,E2 -4581.32} C_VEL
LIN {X 0,Y 523.661,Z 589.669,A -85,B 0,C 180,E1 -4582.481,E2 -4582.481} C_VEL
LIN {X 0,Y 523.528,Z 596.743,A -85,B 0,C 180,E1 -4583.835,E2 -4583.835} C_VEL
LIN {X 0,Y 523.384,Z 601.46,A -85,B 0,C 180,E1 -4584.993,E2 -4584.993} C_VEL
LIN {X 0,Y 523.443,Z 605.069,A -85,B 0,C 180,E1 -4586.151,E2 -4586.151} C_VEL
LIN {X 0,Y 523.367,Z 606.938,A -85,B 0,C 180,E1 -4586.921,E2 -4586.921} C_VEL
LIN {X 0,Y 523.335,Z 608.348,A -85,B 0,C 180,E1 -4587.691,E2 -4587.691} C_VEL
LIN {X 0,Y 523.25,Z 609.968,A -85,B 0,C 180,E1 -4589.231,E2 -4589.231} C_VEL
LIN {X 0,Y 523.247,Z 610.206,A -85,B 0,C 180,E1 -4590,E2 -4590} C_VEL
LIN {X 0,Y 523.25,Z 610.023,A -85,B 0,C 180,E1 -4590.77,E2 -4590.77} C_VEL
LIN {X 0,Y 523.335,Z 608.475,A -85,B 0,C 180,E1 -4592.309,E2 -4592.309} C_VEL
LIN {X 0,Y 523.368,Z 607.12,A -85,B 0,C 180,E1 -4593.079,E2 -4593.079} C_VEL
LIN {X 0,Y 523.442,Z 604.255,A -85,B 0,C 180,E1 -4594.235,E2 -4594.235} C_VEL
LIN {X 0,Y 523.463,Z 600.372,A -85,B 0,C 180,E1 -4595.393,E2 -4595.393} C_VEL
LIN {X 0,Y 523.53,Z 595.198,A -85,B 0,C 180,E1 -4596.587,E2 -4596.587} C_VEL
LIN {X 0,Y 523.728,Z 587.832,A -85,B 0,C 180,E1 -4597.906,E2 -4597.906} C_VEL
LIN {X 0,Y 523.88,Z 579.68,A -85,B 0,C 180,E1 -4599.07,E2 -4599.07} C_VEL
LIN {X 0,Y 524.11,Z 571.335,A -85,B 0,C 180,E1 -4600.039,E2 -4600.039} C_VEL
LIN {X 0,Y 524.426,Z 561.033,A -85,B 0,C 180,E1 -4601.01,E2 -4601.01} C_VEL
LIN {X 0,Y 524.72,Z 549.707,A -85,B 0,C 180,E1 -4601.863,E2 -4601.863} C_VEL
LIN {X 0,Y 524.977,Z 539.665,A -85,B 0,C 180,E1 -4602.467,E2 -4602.467} C_VEL
LIN {X 0,Y 525.193,Z 528.353,A -85,B 0,C 180,E1 -4603.002,E2 -4603.002} C_VEL
LIN {X 0,Y 525.447,Z 515.504,A -85,B 0,C 180,E1 -4603.438,E2 -4603.438} C_VEL
LIN {X 0,Y 525.608,Z 501.823,A -85,B 0,C 180,E1 -4603.73,E2 -4603.73} C_VEL
LIN {X 0,Y 525.9,Z 409.112,A -85,B 0,C 180,E1 -4605.006,E2 -4605.006} C_VEL
LIN {X 0,Y 524.236,Z 399.595,A -85,B 0,C 180,E1 -4605.194,E2 -4605.194} C_VEL
LIN {X 0,Y 524.631,Z 383.042,A -85,B 0,C 180,E1 -4608.309,E2 -4608.309} C_VEL
LIN {X 0,Y 524.784,Z 374.495,A -85,B 0,C 180,E1 -4609.941,E2 -4609.941} C_VEL
LIN {X 0,Y 523.975,Z 368.72,A -85,B 0,C 180,E1 -4611.129,E2 -4611.129} C_VEL
LIN {X 0,Y 523.936,Z 368.726,A -85,B 0,C 180,E1 -4614.572,E2 -4614.572} C_VEL
LIN {X 0,Y 523.953,Z 368.72,A -85,B 0,C 180,E1 -4617.133,E2 -4617.133} C_VEL
LIN {X 0,Y 523.946,Z 368.715,A -85,B 0,C 180,E1 -4619.756,E2 -4619.756} C_VEL
LIN {X 0,Y 523.938,Z 368.72,A -85,B 0,C 180,E1 -4622.45,E2 -4622.45} C_VEL
LIN {X 0,Y 523.928,Z 368.719,A -85,B 0,C 180,E1 -4625.227,E2 -4625.227} C_VEL
LIN {X 0,Y 523.92,Z 368.72,A -85,B 0,C 180,E1 -4628.102,E2 -4628.102} C_VEL
LIN {X 0,Y 523.943,Z 368.718,A -85,B 0,C 180,E1 -4631.092,E2 -4631.092} C_VEL
LIN {X 0,Y 523.941,Z 368.719,A -85,B 0,C 180,E1 -4634.228,E2 -4634.228} C_VEL
LIN {X 0,Y 523.931,Z 368.721,A -85,B 0,C 180,E1 -4636.834,E2 -4636.834} C_VEL
LIN {X 0,Y 523.947,Z 368.718,A -85,B 0,C 180,E1 -4638.908,E2 -4638.908} C_VEL
LIN {X 0,Y 523.919,Z 368.72,A -85,B 0,C 180,E1 -4641.898,E2 -4641.898} C_VEL
LIN {X 0,Y 523.93,Z 368.719,A -85,B 0,C 180,E1 -4644.911,E2 -4644.911} C_VEL
LIN {X 0,Y 523.94,Z 368.716,A -85,B 0,C 180,E1 -4647.68,E2 -4647.68} C_VEL
LIN {X 0,Y 523.96,Z 368.717,A -85,B 0,C 180,E1 -4650.677,E2 -4650.677} C_VEL
LIN {X 0,Y 523.98,Z 368.713,A -85,B 0,C 180,E1 -4653.729,E2 -4653.729} C_VEL
LIN {X 0,Y 523.918,Z 368.727,A -85,B 0,C 180,E1 -4656.27,E2 -4656.27} C_VEL
LIN {X 0,Y 523.952,Z 368.716,A -85,B 0,C 180,E1 -4658.767,E2 -4658.767} C_VEL
LIN {X 0,Y 523.957,Z 368.713,A -85,B 0,C 180,E1 -4661.221,E2 -4661.221} C_VEL
LIN {X 0,Y 523.942,Z 368.718,A -85,B 0,C 180,E1 -4663.639,E2 -4663.639} C_VEL
LIN {X 0,Y 523.947,Z 368.724,A -85,B 0,C 180,E1 -4666.028,E2 -4666.028} C_VEL
LIN {X 0,Y 524.019,Z 368.709,A -85,B 0,C 180,E1 -4668.394,E2 -4668.394} C_VEL
LIN {X 0,Y 524.007,Z 368.71,A -85,B 0,C 180,E1 -4671.516,E2 -4671.516} C_VEL
LIN {X 0,Y 524.088,Z 368.698,A -85,B 0,C 180,E1 -4674.614,E2 -4674.614} C_VEL
LIN {X 0,Y 524.117,Z 368.7,A -85,B 0,C 180,E1 -4677.694,E2 -4677.694} C_VEL
LIN {X 0,Y 524.128,Z 368.692,A -85,B 0,C 180,E1 -4680.768,E2 -4680.768} C_VEL
LIN {X 0,Y 524.078,Z 368.699,A -85,B 0,C 180,E1 -4683.075,E2 -4683.075} C_VEL
LIN {X 0,Y 524.052,Z 368.705,A -85,B 0,C 180,E1 -4686.159,E2 -4686.159} C_VEL
LIN {X 0,Y 523.991,Z 368.712,A -85,B 0,C 180,E1 -4689.262,E2 -4689.262} C_VEL
LIN {X 0,Y 524.031,Z 368.712,A -85,B 0,C 180,E1 -4691.751,E2 -4691.751} C_VEL
LIN {X 0,Y 523.999,Z 368.71,A -85,B 0,C 180,E1 -4695.052,E2 -4695.052} C_VEL
LIN {X 0,Y 523.969,Z 368.715,A -85,B 0,C 180,E1 -4697.969,E2 -4697.969} C_VEL
LIN {X 0,Y 523.978,Z 368.711,A -85,B 0,C 180,E1 -4700.41,E2 -4700.41} C_VEL
LIN {X 0,Y 523.917,Z 368.72,A -85,B 0,C 180,E1 -4702.893,E2 -4702.893} C_VEL
LIN {X 0,Y 523.989,Z 368.711,A -85,B 0,C 180,E1 -4706.019,E2 -4706.019} C_VEL
LIN {X 0,Y 523.943,Z 368.718,A -85,B 0,C 180,E1 -4708.875,E2 -4708.875} C_VEL
LIN {X 0,Y 523.925,Z 368.723,A -85,B 0,C 180,E1 -4711.544,E2 -4711.544} C_VEL
LIN {X 0,Y 523.924,Z 368.717,A -85,B 0,C 180,E1 -4714.291,E2 -4714.291} C_VEL
LIN {X 0,Y 523.911,Z 368.727,A -85,B 0,C 180,E1 -4717.132,E2 -4717.132} C_VEL
LIN {X 0,Y 523.942,Z 368.715,A -85,B 0,C 180,E1 -4720.13,E2 -4720.13} C_VEL
LIN {X 0,Y 523.926,Z 368.726,A -85,B 0,C 180,E1 -4723.167,E2 -4723.167} C_VEL
LIN {X 0,Y 523.94,Z 368.716,A -85,B 0,C 180,E1 -4725.771,E2 -4725.771} C_VEL
LIN {X 0,Y 523.943,Z 368.722,A -85,B 0,C 180,E1 -4728.908,E2 -4728.908} C_VEL
LIN {X 0,Y 523.921,Z 368.718,A -85,B 0,C 180,E1 -4731.898,E2 -4731.898} C_VEL
LIN {X 0,Y 523.934,Z 368.725,A -85,B 0,C 180,E1 -4734.91,E2 -4734.91} C_VEL
LIN {X 0,Y 523.939,Z 368.716,A -85,B 0,C 180,E1 -4737.679,E2 -4737.679} C_VEL
LIN {X 0,Y 523.959,Z 368.721,A -85,B 0,C 180,E1 -4740.676,E2 -4740.676} C_VEL
LIN {X 0,Y 523.978,Z 368.714,A -85,B 0,C 180,E1 -4743.728,E2 -4743.728} C_VEL
LIN {X 0,Y 523.994,Z 368.916,A -85,B 0,C 180,E1 -4746.096,E2 -4746.096} C_VEL
LIN {X 0,Y 525.33,Z 376.292,A -85,B 0,C 180,E1 -4747.384,E2 -4747.384} C_VEL
LIN {X 0,Y 524.958,Z 392.527,A -85,B 0,C 180,E1 -4750.038,E2 -4750.038} C_VEL
LIN {X 0,Y 524.535,Z 410.042,A -85,B 0,C 180,E1 -4752.856,E2 -4752.856} C_VEL
LIN {X 0,Y 524.302,Z 422.522,A -85,B 0,C 180,E1 -4754.845,E2 -4754.845} C_VEL
LIN {X 0,Y 525.963,Z 434.291,A -85,B 0,C 180,E1 -4755.058,E2 -4755.058} C_VEL
LIN {X 0,Y 525.512,Z 530.481,A -85,B 0,C 180,E1 -4756.391,E2 -4756.391} C_VEL
LIN {X 0,Y 525.276,Z 543.768,A -85,B 0,C 180,E1 -4756.73,E2 -4756.73} C_VEL
LIN {X 0,Y 525.032,Z 557.062,A -85,B 0,C 180,E1 -4757.24,E2 -4757.24} C_VEL
LIN {X 0,Y 524.726,Z 569.294,A -85,B 0,C 180,E1 -4757.888,E2 -4757.888} C_VEL
LIN {X 0,Y 524.487,Z 581.113,A -85,B 0,C 180,E1 -4758.698,E2 -4758.698} C_VEL
LIN {X 0,Y 524.208,Z 591.306,A -85,B 0,C 180,E1 -4759.572,E2 -4759.572} C_VEL
LIN {X 0,Y 523.953,Z 600.477,A -85,B 0,C 180,E1 -4760.542,E2 -4760.542} C_VEL
LIN {X 0,Y 523.735,Z 609.413,A -85,B 0,C 180,E1 -4761.706,E2 -4761.706} C_VEL
LIN {X 0,Y 523.584,Z 616.605,A -85,B 0,C 180,E1 -4762.867,E2 -4762.867} C_VEL
LIN {X 0,Y 523.524,Z 623.155,A -85,B 0,C 180,E1 -4764.221,E2 -4764.221} C_VEL
LIN {X 0,Y 523.36,Z 627.484,A -85,B 0,C 180,E1 -4765.378,E2 -4765.378} C_VEL
LIN {X 0,Y 523.443,Z 629.78,A -85,B 0,C 180,E1 -4766.151,E2 -4766.151} C_VEL
LIN {X 0,Y 523.367,Z 631.637,A -85,B 0,C 180,E1 -4766.921,E2 -4766.921} C_VEL
LIN {X 0,Y 523.334,Z 633.03,A -85,B 0,C 180,E1 -4767.691,E2 -4767.691} C_VEL
LIN {X 0,Y 523.25,Z 634.63,A -85,B 0,C 180,E1 -4769.23,E2 -4769.23} C_VEL
LIN {X 0,Y 523.246,Z 634.846,A -85,B 0,C 180,E1 -4770,E2 -4770} C_VEL
LIN {X 0,Y 523.274,Z 634.025,A -85,B 0,C 180,E1 -4771.539,E2 -4771.539} C_VEL
LIN {X 0,Y 523.334,Z 633.034,A -85,B 0,C 180,E1 -4772.309,E2 -4772.309} C_VEL
LIN {X 0,Y 523.367,Z 631.641,A -85,B 0,C 180,E1 -4773.079,E2 -4773.079} C_VEL
LIN {X 0,Y 523.424,Z 628.712,A -85,B 0,C 180,E1 -4774.235,E2 -4774.235} C_VEL
LIN {X 0,Y 523.464,Z 624.745,A -85,B 0,C 180,E1 -4775.393,E2 -4775.393} C_VEL
LIN {X 0,Y 523.519,Z 619.52,A -85,B 0,C 180,E1 -4776.576,E2 -4776.576} C_VEL
LIN {X 0,Y 523.654,Z 613.21,A -85,B 0,C 180,E1 -4777.713,E2 -4777.713} C_VEL
LIN {X 0,Y 523.838,Z 605.188,A -85,B 0,C 180,E1 -4778.875,E2 -4778.875} C_VEL
LIN {X 0,Y 524.064,Z 597.015,A -85,B 0,C 180,E1 -4779.845,E2 -4779.845} C_VEL
LIN {X 0,Y 524.351,Z 587.047,A -85,B 0,C 180,E1 -4780.815,E2 -4780.815} C_VEL
LIN {X 0,Y 524.607,Z 575.813,A -85,B 0,C 180,E1 -4781.689,E2 -4781.689} C_VEL
LIN {X 0,Y 524.916,Z 564.766,A -85,B 0,C 180,E1 -4782.37,E2 -4782.37} C_VEL
LIN {X 0,Y 525.155,Z 552.544,A -85,B 0,C 180,E1 -4782.953,E2 -4782.953} C_VEL
